//     Standard Inputs/MAIN.R7.T02_STAT/SGs_COM_ERR @bit 1 <-> StandardInputs/Standard Out Var 12
//     Standard Inputs/MAIN.R7.T02_STAT/SGs_COM_ERR <-> StandardInputs/Standard Out Var 9
//     Standard Inputs/MAIN.R7.T02_STAT/SGs_FB_ERR @bit 1 <-> StandardInputs/Standard Out Var 11
//     Standard Inputs/MAIN.R7.T02_STAT/SGs_FB_ERR <-> StandardInputs/Standard Out Var 8
//     Standard Inputs/MAIN.R7.T02_STAT/SGs_OUT_ERR <-> StandardInputs/Standard Out Var 10
//     Standard Inputs/MAIN.R7.T02_STAT/SGs_OUT_ERR @bit 1 <-> StandardInputs/Standard Out Var 13
//     Standard Outputs/MAIN.R7.T02_CMD/FBs_ControlPowerPB <-> StandardOutputs/Standard In Var 7
//     Standard Outputs/MAIN.R7.T02_CMD/SGs_ERRAck <-> StandardOutputs/Standard In Var 4
//     Standard Outputs/MAIN.R7.T02_CMD/SGs_ERRAck <-> StandardOutputs/Standard In Var 6
//     Standard Outputs/MAIN.R7.T02_CMD/SGs_RUNSTOP <-> StandardOutputs/Standard In Var 3
//     Standard Outputs/MAIN.R7.T02_CMD/SGs_RUNSTOP <-> StandardOutputs/Standard In Var 5
//     Standard Outputs/MAIN.Safety_Zone_Test <-> StandardOutputs/Standard In Var 21
//   SODG11_SSCC610_2403701_PLC/SODG11_SSCC610_2403701_PLC Instance <-> EtherCAT Master (EtherCAT)/R7.T01 (EK1100)/R7.T03 (EL1904)
//     Standard Inputs/MAIN.R7.T03/I <-> Module 1 (FSOES)/TxPDO/FSOE/InputChannel1
//     Standard Inputs/MAIN.R7.T03/I @bit 1 <-> Module 1 (FSOES)/TxPDO/FSOE/InputChannel2
//     Standard Inputs/MAIN.R7.T03/I @bit 2 <-> Module 1 (FSOES)/TxPDO/FSOE/InputChannel3
//     Standard Inputs/MAIN.R7.T03/I @bit 3 <-> Module 1 (FSOES)/TxPDO/FSOE/InputChannel4
//     Standard Inputs/MAIN.R7.T03/InfoData/State <-> InfoData/State
//   SODG11_SSCC610_2403701_PLC/SODG11_SSCC610_2403701_PLC Instance <-> EtherCAT Master (EtherCAT)/R7.T01 (EK1100)/R7.T04 (EK1122)
//     Standard Inputs/MAIN.R7.T04/InfoData/State <-> InfoData/State
//   SODG11_SSCC610_2403701_PLC/SODG11_SSCC610_2403701_PLC Instance <-> EtherCAT Master (EtherCAT)/R7.T01 (EK1100)/R7.T04 (EK1122)/R7.Reamer[1].N01 (EP1008-0002)
//     Standard Inputs/MAIN.R7.Reamer[1].N01/I <-> Channel 1/Input
//     Standard Inputs/MAIN.R7.Reamer[1].N01/I @bit 1 <-> Channel 2/Input
//     Standard Inputs/MAIN.R7.Reamer[1].N01/I @bit 2 <-> Channel 3/Input
//     Standard Inputs/MAIN.R7.Reamer[1].N01/I @bit 3 <-> Channel 4/Input
//     Standard Inputs/MAIN.R7.Reamer[1].N01/I @bit 4 <-> Channel 5/Input
//     Standard Inputs/MAIN.R7.Reamer[1].N01/I @bit 5 <-> Channel 6/Input
//     Standard Inputs/MAIN.R7.Reamer[1].N01/I @bit 6 <-> Channel 7/Input
//     Standard Inputs/MAIN.R7.Reamer[1].N01/I @bit 7 <-> Channel 8/Input
//     Standard Inputs/MAIN.R7.Reamer[1].N01/InfoData/State <-> InfoData/State
//     Standard Inputs/MAIN.R7.Reamer[1].N01/Wc_State <-> WcState/WcState
//   SODG11_SSCC610_2403701_PLC/SODG11_SSCC610_2403701_PLC Instance <-> EtherCAT Master (EtherCAT)/R7.T01 (EK1100)/R7.T04 (EK1122)/R7.Reamer[1].N30 (EP2028-0002)
//     Standard Inputs/MAIN.R7.Reamer[1].N30_STAT/InfoData/State <-> InfoData/State
//     Standard Outputs/MAIN.R7.Reamer[1].N30/Q <-> Channel 1/Output
//     Standard Outputs/MAIN.R7.Reamer[1].N30/Q @bit {1..7} <-> Channel {2..8}/Output  (7 links)
//   SODG11_SSCC610_2403701_PLC/SODG11_SSCC610_2403701_PLC Instance <-> EtherCAT Master (EtherCAT)/R8.RT02 (EL6695-1001)
//     Standard Inputs/MAIN.R8.In_From_HW/BYTE_[10] <-> Module 3 (Default IO)/Std. In (64 Bytes)/Input DWORD 2 @bit 8
//     Standard Inputs/MAIN.R8.In_From_HW/BYTE_[11] <-> Module 3 (Default IO)/Std. In (64 Bytes)/Input DWORD 2 @bit 16
//     Standard Inputs/MAIN.R8.In_From_HW/BYTE_[12] <-> Module 3 (Default IO)/Std. In (64 Bytes)/Input DWORD 2 @bit 24
//     Standard Inputs/MAIN.R8.In_From_HW/BYTE_[14] <-> Module 3 (Default IO)/Std. In (64 Bytes)/Input DWORD 3 @bit 8
//     Standard Inputs/MAIN.R8.In_From_HW/BYTE_[15] <-> Module 3 (Default IO)/Std. In (64 Bytes)/Input DWORD 3 @bit 16
//     Standard Inputs/MAIN.R8.In_From_HW/BYTE_[16] <-> Module 3 (Default IO)/Std. In (64 Bytes)/Input DWORD 3 @bit 24
//     Standard Inputs/MAIN.R8.In_From_HW/BYTE_[18] <-> Module 3 (Default IO)/Std. In (64 Bytes)/Input DWORD 4 @bit 8
//     Standard Inputs/MAIN.R8.In_From_HW/BYTE_[19] <-> Module 3 (Default IO)/Std. In (64 Bytes)/Input DWORD 4 @bit 16
//     Standard Inputs/MAIN.R8.In_From_HW/BYTE_[20] <-> Module 3 (Default IO)/Std. In (64 Bytes)/Input DWORD 4 @bit 24
//     Standard Inputs/MAIN.R8.In_From_HW/BYTE_[22] <-> Module 3 (Default IO)/Std. In (64 Bytes)/Input DWORD 5 @bit 8
//     Standard Inputs/MAIN.R8.In_From_HW/BYTE_[23] <-> Module 3 (Default IO)/Std. In (64 Bytes)/Input DWORD 5 @bit 16
//     Standard Inputs/MAIN.R8.In_From_HW/BYTE_[24] <-> Module 3 (Default IO)/Std. In (64 Bytes)/Input DWORD 5 @bit 24
//     Standard Inputs/MAIN.R8.In_From_HW/BYTE_[26] <-> Module 3 (Default IO)/Std. In (64 Bytes)/Input DWORD 6 @bit 8
//     Standard Inputs/MAIN.R8.In_From_HW/BYTE_[27] <-> Module 3 (Default IO)/Std. In (64 Bytes)/Input DWORD 6 @bit 16
//     Standard Inputs/MAIN.R8.In_From_HW/BYTE_[28] <-> Module 3 (Default IO)/Std. In (64 Bytes)/Input DWORD 6 @bit 24
//     Standard Inputs/MAIN.R8.In_From_HW/BYTE_[2] <-> Module 3 (Default IO)/Std. In (64 Bytes)/Input DWORD 0 @bit 8
//     Standard Inputs/MAIN.R8.In_From_HW/BYTE_[30] <-> Module 3 (Default IO)/Std. In (64 Bytes)/Input DWORD 7 @bit 8
//     Standard Inputs/MAIN.R8.In_From_HW/BYTE_[31] <-> Module 3 (Default IO)/Std. In (64 Bytes)/Input DWORD 7 @bit 16
//     Standard Inputs/MAIN.R8.In_From_HW/BYTE_[32] <-> Module 3 (Default IO)/Std. In (64 Bytes)/Input DWORD 7 @bit 24
//     Standard Inputs/MAIN.R8.In_From_HW/BYTE_[34] <-> Module 3 (Default IO)/Std. In (64 Bytes)/Input DWORD 8 @bit 8
//     Standard Inputs/MAIN.R8.In_From_HW/BYTE_[35] <-> Module 3 (Default IO)/Std. In (64 Bytes)/Input DWORD 8 @bit 16
//     Standard Inputs/MAIN.R8.In_From_HW/BYTE_[36] <-> Module 3 (Default IO)/Std. In (64 Bytes)/Input DWORD 8 @bit 24
//     Standard Inputs/MAIN.R8.In_From_HW/BYTE_[38] <-> Module 3 (Default IO)/Std. In (64 Bytes)/Input DWORD 9 @bit 8
//     Standard Inputs/MAIN.R8.In_From_HW/BYTE_[39] <-> Module 3 (Default IO)/Std. In (64 Bytes)/Input DWORD 9 @bit 16
//     Standard Inputs/MAIN.R8.In_From_HW/BYTE_[3] <-> Module 3 (Default IO)/Std. In (64 Bytes)/Input DWORD 0 @bit 16
//     Standard Inputs/MAIN.R8.In_From_HW/BYTE_[40] <-> Module 3 (Default IO)/Std. In (64 Bytes)/Input DWORD 9 @bit 24
//     Standard Inputs/MAIN.R8.In_From_HW/BYTE_[42] <-> Module 3 (Default IO)/Std. In (64 Bytes)/Input DWORD 10 @bit 8
//     Standard Inputs/MAIN.R8.In_From_HW/BYTE_[43] <-> Module 3 (Default IO)/Std. In (64 Bytes)/Input DWORD 10 @bit 16
//     Standard Inputs/MAIN.R8.In_From_HW/BYTE_[44] <-> Module 3 (Default IO)/Std. In (64 Bytes)/Input DWORD 10 @bit 24
//     Standard Inputs/MAIN.R8.In_From_HW/BYTE_[46] <-> Module 3 (Default IO)/Std. In (64 Bytes)/Input DWORD 11 @bit 8
//     Standard Inputs/MAIN.R8.In_From_HW/BYTE_[47] <-> Module 3 (Default IO)/Std. In (64 Bytes)/Input DWORD 11 @bit 16
//     Standard Inputs/MAIN.R8.In_From_HW/BYTE_[48] <-> Module 3 (Default IO)/Std. In (64 Bytes)/Input DWORD 11 @bit 24
//     Standard Inputs/MAIN.R8.In_From_HW/BYTE_[4] <-> Module 3 (Default IO)/Std. In (64 Bytes)/Input DWORD 0 @bit 24
//     Standard Inputs/MAIN.R8.In_From_HW/BYTE_[50] <-> Module 3 (Default IO)/Std. In (64 Bytes)/Input DWORD 12 @bit 8
//     Standard Inputs/MAIN.R8.In_From_HW/BYTE_[51] <-> Module 3 (Default IO)/Std. In (64 Bytes)/Input DWORD 12 @bit 16
//     Standard Inputs/MAIN.R8.In_From_HW/BYTE_[52] <-> Module 3 (Default IO)/Std. In (64 Bytes)/Input DWORD 12 @bit 24
//     Standard Inputs/MAIN.R8.In_From_HW/BYTE_[54] <-> Module 3 (Default IO)/Std. In (64 Bytes)/Input DWORD 13 @bit 8
//     Standard Inputs/MAIN.R8.In_From_HW/BYTE_[55] <-> Module 3 (Default IO)/Std. In (64 Bytes)/Input DWORD 13 @bit 16
//     Standard Inputs/MAIN.R8.In_From_HW/BYTE_[56] <-> Module 3 (Default IO)/Std. In (64 Bytes)/Input DWORD 13 @bit 24
//     Standard Inputs/MAIN.R8.In_From_HW/BYTE_[58] <-> Module 3 (Default IO)/Std. In (64 Bytes)/Input DWORD 14 @bit 8
//     Standard Inputs/MAIN.R8.In_From_HW/BYTE_[59] <-> Module 3 (Default IO)/Std. In (64 Bytes)/Input DWORD 14 @bit 16
//     Standard Inputs/MAIN.R8.In_From_HW/BYTE_[60] <-> Module 3 (Default IO)/Std. In (64 Bytes)/Input DWORD 14 @bit 24
//     Standard Inputs/MAIN.R8.In_From_HW/BYTE_[62] <-> Module 3 (Default IO)/Std. In (64 Bytes)/Input DWORD 15 @bit 8
//     Standard Inputs/MAIN.R8.In_From_HW/BYTE_[63] <-> Module 3 (Default IO)/Std. In (64 Bytes)/Input DWORD 15 @bit 16
//     Standard Inputs/MAIN.R8.In_From_HW/BYTE_[64] <-> Module 3 (Default IO)/Std. In (64 Bytes)/Input DWORD 15 @bit 24
//     Standard Inputs/MAIN.R8.In_From_HW/BYTE_[6] <-> Module 3 (Default IO)/Std. In (64 Bytes)/Input DWORD 1 @bit 8
//     Standard Inputs/MAIN.R8.In_From_HW/BYTE_[7] <-> Module 3 (Default IO)/Std. In (64 Bytes)/Input DWORD 1 @bit 16
//     Standard Inputs/MAIN.R8.In_From_HW/BYTE_[8] <-> Module 3 (Default IO)/Std. In (64 Bytes)/Input DWORD 1 @bit 24
//     Standard Inputs/MAIN.R8.In_From_HW/BYTE_[{1..61 step 4}] <-> Module 3 (Default IO)/Std. In (64 Bytes)/Input DWORD {0..15}  (16 links)
//     Standard Inputs/MAIN.R8.RT02/External_device_not_connected <-> Module 1 (Sync Inputs)/Compact/External device not connected
//     Standard Inputs/MAIN.R8.RT02/FSOE_Inputs_ConnID <-> Module 2 (Safety Data (8 Byte))/Inputs/FSOE/FSOE ConnID
//     Standard Inputs/MAIN.R8.RT02/FSOE_Inputs_Data_0 <-> Module 2 (Safety Data (8 Byte))/Inputs/FSOE/FSOE Data_0
//     Standard Inputs/MAIN.R8.RT02/FSOE_Inputs_Data_1 <-> Module 2 (Safety Data (8 Byte))/Inputs/FSOE/FSOE Data_1
//     Standard Inputs/MAIN.R8.RT02/FSOE_Inputs_Data_2 <-> Module 2 (Safety Data (8 Byte))/Inputs/FSOE/FSOE Data_2
//     Standard Inputs/MAIN.R8.RT02/FSOE_Inputs_Data_3 <-> Module 2 (Safety Data (8 Byte))/Inputs/FSOE/FSOE Data_3
//     Standard Inputs/MAIN.R8.RT02/InfoData/AdsAddr/netId <-> InfoData/AdsAddr/netId
//     Standard Inputs/MAIN.R8.RT02/InfoData/AdsAddr/port <-> InfoData/AdsAddr/port
//     Standard Inputs/MAIN.R8.RT02/InfoData/State <-> InfoData/State
//     Standard Inputs/MAIN.R8.RT02/TxPDO_State <-> Module 1 (Sync Inputs)/Compact/TxPDO state
//     Standard Inputs/MAIN.R8.RT02/TxPDO_Toogle <-> Module 1 (Sync Inputs)/Compact/TxPDO toggle
//     Standard Outputs/MAIN.R8.Out_To_HW/Byte_[10] <-> Module 3 (Default IO)/Std. Out (64 Bytes)/Output DWORD 2 @bit 8
//     Standard Outputs/MAIN.R8.Out_To_HW/Byte_[11] <-> Module 3 (Default IO)/Std. Out (64 Bytes)/Output DWORD 2 @bit 16
//     Standard Outputs/MAIN.R8.Out_To_HW/Byte_[12] <-> Module 3 (Default IO)/Std. Out (64 Bytes)/Output DWORD 2 @bit 24
//     Standard Outputs/MAIN.R8.Out_To_HW/Byte_[14] <-> Module 3 (Default IO)/Std. Out (64 Bytes)/Output DWORD 3 @bit 8
//     Standard Outputs/MAIN.R8.Out_To_HW/Byte_[15] <-> Module 3 (Default IO)/Std. Out (64 Bytes)/Output DWORD 3 @bit 16
//     Standard Outputs/MAIN.R8.Out_To_HW/Byte_[16] <-> Module 3 (Default IO)/Std. Out (64 Bytes)/Output DWORD 3 @bit 24
//     Standard Outputs/MAIN.R8.Out_To_HW/Byte_[18] <-> Module 3 (Default IO)/Std. Out (64 Bytes)/Output DWORD 4 @bit 8
//     Standard Outputs/MAIN.R8.Out_To_HW/Byte_[19] <-> Module 3 (Default IO)/Std. Out (64 Bytes)/Output DWORD 4 @bit 16
//     Standard Outputs/MAIN.R8.Out_To_HW/Byte_[20] <-> Module 3 (Default IO)/Std. Out (64 Bytes)/Output DWORD 4 @bit 24
//     Standard Outputs/MAIN.R8.Out_To_HW/Byte_[22] <-> Module 3 (Default IO)/Std. Out (64 Bytes)/Output DWORD 5 @bit 8
//     Standard Outputs/MAIN.R8.Out_To_HW/Byte_[23] <-> Module 3 (Default IO)/Std. Out (64 Bytes)/Output DWORD 5 @bit 16
//     Standard Outputs/MAIN.R8.Out_To_HW/Byte_[24] <-> Module 3 (Default IO)/Std. Out (64 Bytes)/Output DWORD 5 @bit 24
//     Standard Outputs/MAIN.R8.Out_To_HW/Byte_[26] <-> Module 3 (Default IO)/Std. Out (64 Bytes)/Output DWORD 6 @bit 8
//     Standard Outputs/MAIN.R8.Out_To_HW/Byte_[27] <-> Module 3 (Default IO)/Std. Out (64 Bytes)/Output DWORD 6 @bit 16
//     Standard Outputs/MAIN.R8.Out_To_HW/Byte_[28] <-> Module 3 (Default IO)/Std. Out (64 Bytes)/Output DWORD 6 @bit 24
//     Standard Outputs/MAIN.R8.Out_To_HW/Byte_[2] <-> Module 3 (Default IO)/Std. Out (64 Bytes)/Output DWORD 0 @bit 8
//     Standard Outputs/MAIN.R8.Out_To_HW/Byte_[30] <-> Module 3 (Default IO)/Std. Out (64 Bytes)/Output DWORD 7 @bit 8
//     Standard Outputs/MAIN.R8.Out_To_HW/Byte_[31] <-> Module 3 (Default IO)/Std. Out (64 Bytes)/Output DWORD 7 @bit 16
//     Standard Outputs/MAIN.R8.Out_To_HW/Byte_[32] <-> Module 3 (Default IO)/Std. Out (64 Bytes)/Output DWORD 7 @bit 24
//     Standard Outputs/MAIN.R8.Out_To_HW/Byte_[34] <-> Module 3 (Default IO)/Std. Out (64 Bytes)/Output DWORD 8 @bit 8
//     Standard Outputs/MAIN.R8.Out_To_HW/Byte_[35] <-> Module 3 (Default IO)/Std. Out (64 Bytes)/Output DWORD 8 @bit 16
//     Standard Outputs/MAIN.R8.Out_To_HW/Byte_[36] <-> Module 3 (Default IO)/Std. Out (64 Bytes)/Output DWORD 8 @bit 24
//     Standard Outputs/MAIN.R8.Out_To_HW/Byte_[38] <-> Module 3 (Default IO)/Std. Out (64 Bytes)/Output DWORD 9 @bit 8
//     Standard Outputs/MAIN.R8.Out_To_HW/Byte_[39] <-> Module 3 (Default IO)/Std. Out (64 Bytes)/Output DWORD 9 @bit 16
//     Standard Outputs/MAIN.R8.Out_To_HW/Byte_[3] <-> Module 3 (Default IO)/Std. Out (64 Bytes)/Output DWORD 0 @bit 16
//     Standard Outputs/MAIN.R8.Out_To_HW/Byte_[40] <-> Module 3 (Default IO)/Std. Out (64 Bytes)/Output DWORD 9 @bit 24
//     Standard Outputs/MAIN.R8.Out_To_HW/Byte_[42] <-> Module 3 (Default IO)/Std. Out (64 Bytes)/Output DWORD 10 @bit 8
//     Standard Outputs/MAIN.R8.Out_To_HW/Byte_[43] <-> Module 3 (Default IO)/Std. Out (64 Bytes)/Output DWORD 10 @bit 16
//     Standard Outputs/MAIN.R8.Out_To_HW/Byte_[44] <-> Module 3 (Default IO)/Std. Out (64 Bytes)/Output DWORD 10 @bit 24
//     Standard Outputs/MAIN.R8.Out_To_HW/Byte_[46] <-> Module 3 (Default IO)/Std. Out (64 Bytes)/Output DWORD 11 @bit 8
//     Standard Outputs/MAIN.R8.Out_To_HW/Byte_[47] <-> Module 3 (Default IO)/Std. Out (64 Bytes)/Output DWORD 11 @bit 16
//     Standard Outputs/MAIN.R8.Out_To_HW/Byte_[48] <-> Module 3 (Default IO)/Std. Out (64 Bytes)/Output DWORD 11 @bit 24
//     Standard Outputs/MAIN.R8.Out_To_HW/Byte_[4] <-> Module 3 (Default IO)/Std. Out (64 Bytes)/Output DWORD 0 @bit 24
//     Standard Outputs/MAIN.R8.Out_To_HW/Byte_[50] <-> Module 3 (Default IO)/Std. Out (64 Bytes)/Output DWORD 12 @bit 8
//     Standard Outputs/MAIN.R8.Out_To_HW/Byte_[51] <-> Module 3 (Default IO)/Std. Out (64 Bytes)/Output DWORD 12 @bit 16
//     Standard Outputs/MAIN.R8.Out_To_HW/Byte_[52] <-> Module 3 (Default IO)/Std. Out (64 Bytes)/Output DWORD 12 @bit 24
//     Standard Outputs/MAIN.R8.Out_To_HW/Byte_[54] <-> Module 3 (Default IO)/Std. Out (64 Bytes)/Output DWORD 13 @bit 8
//     Standard Outputs/MAIN.R8.Out_To_HW/Byte_[55] <-> Module 3 (Default IO)/Std. Out (64 Bytes)/Output DWORD 13 @bit 16
//     Standard Outputs/MAIN.R8.Out_To_HW/Byte_[56] <-> Module 3 (Default IO)/Std. Out (64 Bytes)/Output DWORD 13 @bit 24
//     Standard Outputs/MAIN.R8.Out_To_HW/Byte_[58] <-> Module 3 (Default IO)/Std. Out (64 Bytes)/Output DWORD 14 @bit 8
//     Standard Outputs/MAIN.R8.Out_To_HW/Byte_[59] <-> Module 3 (Default IO)/Std. Out (64 Bytes)/Output DWORD 14 @bit 16
//     Standard Outputs/MAIN.R8.Out_To_HW/Byte_[60] <-> Module 3 (Default IO)/Std. Out (64 Bytes)/Output DWORD 14 @bit 24
//     Standard Outputs/MAIN.R8.Out_To_HW/Byte_[62] <-> Module 3 (Default IO)/Std. Out (64 Bytes)/Output DWORD 15 @bit 8
//     Standard Outputs/MAIN.R8.Out_To_HW/Byte_[63] <-> Module 3 (Default IO)/Std. Out (64 Bytes)/Output DWORD 15 @bit 16
//     Standard Outputs/MAIN.R8.Out_To_HW/Byte_[64] <-> Module 3 (Default IO)/Std. Out (64 Bytes)/Output DWORD 15 @bit 24
//     Standard Outputs/MAIN.R8.Out_To_HW/Byte_[6] <-> Module 3 (Default IO)/Std. Out (64 Bytes)/Output DWORD 1 @bit 8
//     Standard Outputs/MAIN.R8.Out_To_HW/Byte_[7] <-> Module 3 (Default IO)/Std. Out (64 Bytes)/Output DWORD 1 @bit 16
//     Standard Outputs/MAIN.R8.Out_To_HW/Byte_[8] <-> Module 3 (Default IO)/Std. Out (64 Bytes)/Output DWORD 1 @bit 24
//     Standard Outputs/MAIN.R8.Out_To_HW/Byte_[{1..61 step 4}] <-> Module 3 (Default IO)/Std. Out (64 Bytes)/Output DWORD {0..15}  (16 links)
//   SODG11_SSCC610_2403701_PLC/SODG11_SSCC610_2403701_PLC Instance <-> EtherCAT Master (EtherCAT)/R8.T01 (EK1100)
//     Standard Inputs/MAIN.R8.T01/InfoData/State <-> InfoData/State
//   SODG11_SSCC610_2403701_PLC/SODG11_SSCC610_2403701_PLC Instance <-> EtherCAT Master (EtherCAT)/R8.T01 (EK1100)/R8.T02 (EL6900)
//     Standard Inputs/MAIN.R8.RT02/FSOE_Outputs_Data_0 @bit 1 <-> StandardInputs/Standard Out Var 14
//     Standard Inputs/MAIN.R8.RT02/FSOE_Outputs_Data_0 @bit 2 <-> StandardInputs/Standard Out Var 15
//     Standard Inputs/MAIN.R8.RT02/FSOE_Outputs_Data_2 @bit 1 <-> StandardInputs/Standard Out Var 18
//     Standard Inputs/MAIN.R8.RT02/FSOE_Outputs_Data_2 <-> StandardInputs/Standard Out Var 17
//     Standard Inputs/MAIN.R8.T02_STAT/Device_Info_Data/Project_CRC <-> Device Info Data/Project CRC
//     Standard Inputs/MAIN.R8.T02_STAT/FBs_FB_ERR <-> StandardInputs/Standard Out Var 16
//     Standard Inputs/MAIN.R8.T02_STAT/FBs_FB_ERR @bit 16 <-> StandardInputs/Standard Out Var 19
//     Standard Inputs/MAIN.R8.T02_STAT/FBs_FB_ERR @bit 29 <-> StandardInputs/Standard Out Var 20
//     Standard Inputs/MAIN.R8.T02_STAT/InfoData/AdsAddr/netId <-> InfoData/AdsAddr/netId
//     Standard Inputs/MAIN.R8.T02_STAT/InfoData/AdsAddr/port <-> InfoData/AdsAddr/port
//     Standard Inputs/MAIN.R8.T02_STAT/InfoData/State <-> InfoData/State
//     Standard Inputs/MAIN.R8.T02_STAT/SGs_COM_ERR @bit 1 <-> StandardInputs/Standard Out Var 12
//     Standard Inputs/MAIN.R8.T02_STAT/SGs_COM_ERR <-> StandardInputs/Standard Out Var 9
//     Standard Inputs/MAIN.R8.T02_STAT/SGs_FB_ERR @bit 1 <-> StandardInputs/Standard Out Var 11
//     Standard Inputs/MAIN.R8.T02_STAT/SGs_FB_ERR <-> StandardInputs/Standard Out Var 8
//     Standard Inputs/MAIN.R8.T02_STAT/SGs_OUT_ERR <-> StandardInputs/Standard Out Var 10
//     Standard Inputs/MAIN.R8.T02_STAT/SGs_OUT_ERR @bit 1 <-> StandardInputs/Standard Out Var 13
//     Standard Outputs/MAIN.R8.T02_CMD/FBs_ControlPowerPB <-> StandardOutputs/Standard In Var 7
//     Standard Outputs/MAIN.R8.T02_CMD/SGs_ERRAck <-> StandardOutputs/Standard In Var 4
//     Standard Outputs/MAIN.R8.T02_CMD/SGs_ERRAck <-> StandardOutputs/Standard In Var 6
//     Standard Outputs/MAIN.R8.T02_CMD/SGs_RUNSTOP <-> StandardOutputs/Standard In Var 3
//     Standard Outputs/MAIN.R8.T02_CMD/SGs_RUNSTOP <-> StandardOutputs/Standard In Var 5
//     Standard Outputs/MAIN.Safety_Zone_Test <-> StandardOutputs/Standard In Var 21
//   SODG11_SSCC610_2403701_PLC/SODG11_SSCC610_2403701_PLC Instance <-> EtherCAT Master (EtherCAT)/R8.T01 (EK1100)/R8.T03 (EL1904)
//     Standard Inputs/MAIN.R8.T03/I <-> Module 1 (FSOES)/TxPDO/FSOE/InputChannel1
//     Standard Inputs/MAIN.R8.T03/I @bit 1 <-> Module 1 (FSOES)/TxPDO/FSOE/InputChannel2
//     Standard Inputs/MAIN.R8.T03/I @bit 2 <-> Module 1 (FSOES)/TxPDO/FSOE/InputChannel3
//     Standard Inputs/MAIN.R8.T03/I @bit 3 <-> Module 1 (FSOES)/TxPDO/FSOE/InputChannel4
//     Standard Inputs/MAIN.R8.T03/InfoData/State <-> InfoData/State
//   SODG11_SSCC610_2403701_PLC/SODG11_SSCC610_2403701_PLC Instance <-> EtherCAT Master (EtherCAT)/R8.T01 (EK1100)/R8.T04 (EK1122)
//     Standard Inputs/MAIN.R8.T04/InfoData/State <-> InfoData/State
//   SODG11_SSCC610_2403701_PLC/SODG11_SSCC610_2403701_PLC Instance <-> EtherCAT Master (EtherCAT)/R8.T01 (EK1100)/R8.T04 (EK1122)/R8.Reamer[1].N01 (EP1008-0002)
//     Standard Inputs/MAIN.R8.Reamer[1].N01/I <-> Channel 1/Input
//     Standard Inputs/MAIN.R8.Reamer[1].N01/I @bit 1 <-> Channel 2/Input
//     Standard Inputs/MAIN.R8.Reamer[1].N01/I @bit 2 <-> Channel 3/Input
//     Standard Inputs/MAIN.R8.Reamer[1].N01/I @bit 3 <-> Channel 4/Input
//     Standard Inputs/MAIN.R8.Reamer[1].N01/I @bit 4 <-> Channel 5/Input
//     Standard Inputs/MAIN.R8.Reamer[1].N01/I @bit 5 <-> Channel 6/Input
//     Standard Inputs/MAIN.R8.Reamer[1].N01/I @bit 6 <-> Channel 7/Input
//     Standard Inputs/MAIN.R8.Reamer[1].N01/I @bit 7 <-> Channel 8/Input
//     Standard Inputs/MAIN.R8.Reamer[1].N01/InfoData/State <-> InfoData/State
//     Standard Inputs/MAIN.R8.Reamer[1].N01/Wc_State <-> WcState/WcState
//   SODG11_SSCC610_2403701_PLC/SODG11_SSCC610_2403701_PLC Instance <-> EtherCAT Master (EtherCAT)/R8.T01 (EK1100)/R8.T04 (EK1122)/R8.Reamer[1].N30 (EP2028-0002)
//     Standard Inputs/MAIN.R8.Reamer[1].N30_STAT/InfoData/State <-> InfoData/State
//     Standard Outputs/MAIN.R8.Reamer[1].N30/Q <-> Channel 1/Output
//     Standard Outputs/MAIN.R8.Reamer[1].N30/Q @bit {1..7} <-> Channel {2..8}/Output  (7 links)
//   SODG11_SSCC610_2403701_PLC/SODG11_SSCC610_2403701_PLC Instance <-> EtherCAT Master (EtherCAT)/R9.RT02 (EL6695-1001)
//     Standard Inputs/MAIN.R9.In_From_HW/BYTE_[10] <-> Module 3 (Default IO)/Std. In (64 Bytes)/Input DWORD 2 @bit 8
//     Standard Inputs/MAIN.R9.In_From_HW/BYTE_[11] <-> Module 3 (Default IO)/Std. In (64 Bytes)/Input DWORD 2 @bit 16
//     Standard Inputs/MAIN.R9.In_From_HW/BYTE_[12] <-> Module 3 (Default IO)/Std. In (64 Bytes)/Input DWORD 2 @bit 24
//     Standard Inputs/MAIN.R9.In_From_HW/BYTE_[14] <-> Module 3 (Default IO)/Std. In (64 Bytes)/Input DWORD 3 @bit 8
//     Standard Inputs/MAIN.R9.In_From_HW/BYTE_[15] <-> Module 3 (Default IO)/Std. In (64 Bytes)/Input DWORD 3 @bit 16
//     Standard Inputs/MAIN.R9.In_From_HW/BYTE_[16] <-> Module 3 (Default IO)/Std. In (64 Bytes)/Input DWORD 3 @bit 24
//     Standard Inputs/MAIN.R9.In_From_HW/BYTE_[18] <-> Module 3 (Default IO)/Std. In (64 Bytes)/Input DWORD 4 @bit 8
//     Standard Inputs/MAIN.R9.In_From_HW/BYTE_[19] <-> Module 3 (Default IO)/Std. In (64 Bytes)/Input DWORD 4 @bit 16
//     Standard Inputs/MAIN.R9.In_From_HW/BYTE_[20] <-> Module 3 (Default IO)/Std. In (64 Bytes)/Input DWORD 4 @bit 24
//     Standard Inputs/MAIN.R9.In_From_HW/BYTE_[22] <-> Module 3 (Default IO)/Std. In (64 Bytes)/Input DWORD 5 @bit 8
//     Standard Inputs/MAIN.R9.In_From_HW/BYTE_[23] <-> Module 3 (Default IO)/Std. In (64 Bytes)/Input DWORD 5 @bit 16
//     Standard Inputs/MAIN.R9.In_From_HW/BYTE_[24] <-> Module 3 (Default IO)/Std. In (64 Bytes)/Input DWORD 5 @bit 24
//     Standard Inputs/MAIN.R9.In_From_HW/BYTE_[26] <-> Module 3 (Default IO)/Std. In (64 Bytes)/Input DWORD 6 @bit 8
//     Standard Inputs/MAIN.R9.In_From_HW/BYTE_[27] <-> Module 3 (Default IO)/Std. In (64 Bytes)/Input DWORD 6 @bit 16
//     Standard Inputs/MAIN.R9.In_From_HW/BYTE_[28] <-> Module 3 (Default IO)/Std. In (64 Bytes)/Input DWORD 6 @bit 24
//     Standard Inputs/MAIN.R9.In_From_HW/BYTE_[2] <-> Module 3 (Default IO)/Std. In (64 Bytes)/Input DWORD 0 @bit 8
//     Standard Inputs/MAIN.R9.In_From_HW/BYTE_[30] <-> Module 3 (Default IO)/Std. In (64 Bytes)/Input DWORD 7 @bit 8
//     Standard Inputs/MAIN.R9.In_From_HW/BYTE_[31] <-> Module 3 (Default IO)/Std. In (64 Bytes)/Input DWORD 7 @bit 16
//     Standard Inputs/MAIN.R9.In_From_HW/BYTE_[32] <-> Module 3 (Default IO)/Std. In (64 Bytes)/Input DWORD 7 @bit 24
//     Standard Inputs/MAIN.R9.In_From_HW/BYTE_[34] <-> Module 3 (Default IO)/Std. In (64 Bytes)/Input DWORD 8 @bit 8
//     Standard Inputs/MAIN.R9.In_From_HW/BYTE_[35] <-> Module 3 (Default IO)/Std. In (64 Bytes)/Input DWORD 8 @bit 16
//     Standard Inputs/MAIN.R9.In_From_HW/BYTE_[36] <-> Module 3 (Default IO)/Std. In (64 Bytes)/Input DWORD 8 @bit 24
//     Standard Inputs/MAIN.R9.In_From_HW/BYTE_[38] <-> Module 3 (Default IO)/Std. In (64 Bytes)/Input DWORD 9 @bit 8
//     Standard Inputs/MAIN.R9.In_From_HW/BYTE_[39] <-> Module 3 (Default IO)/Std. In (64 Bytes)/Input DWORD 9 @bit 16
//     Standard Inputs/MAIN.R9.In_From_HW/BYTE_[3] <-> Module 3 (Default IO)/Std. In (64 Bytes)/Input DWORD 0 @bit 16
//     Standard Inputs/MAIN.R9.In_From_HW/BYTE_[40] <-> Module 3 (Default IO)/Std. In (64 Bytes)/Input DWORD 9 @bit 24
//     Standard Inputs/MAIN.R9.In_From_HW/BYTE_[42] <-> Module 3 (Default IO)/Std. In (64 Bytes)/Input DWORD 10 @bit 8
//     Standard Inputs/MAIN.R9.In_From_HW/BYTE_[43] <-> Module 3 (Default IO)/Std. In (64 Bytes)/Input DWORD 10 @bit 16
//     Standard Inputs/MAIN.R9.In_From_HW/BYTE_[44] <-> Module 3 (Default IO)/Std. In (64 Bytes)/Input DWORD 10 @bit 24
//     Standard Inputs/MAIN.R9.In_From_HW/BYTE_[46] <-> Module 3 (Default IO)/Std. In (64 Bytes)/Input DWORD 11 @bit 8
//     Standard Inputs/MAIN.R9.In_From_HW/BYTE_[47] <-> Module 3 (Default IO)/Std. In (64 Bytes)/Input DWORD 11 @bit 16
//     Standard Inputs/MAIN.R9.In_From_HW/BYTE_[48] <-> Module 3 (Default IO)/Std. In (64 Bytes)/Input DWORD 11 @bit 24
//     Standard Inputs/MAIN.R9.In_From_HW/BYTE_[4] <-> Module 3 (Default IO)/Std. In (64 Bytes)/Input DWORD 0 @bit 24
//     Standard Inputs/MAIN.R9.In_From_HW/BYTE_[50] <-> Module 3 (Default IO)/Std. In (64 Bytes)/Input DWORD 12 @bit 8
//     Standard Inputs/MAIN.R9.In_From_HW/BYTE_[51] <-> Module 3 (Default IO)/Std. In (64 Bytes)/Input DWORD 12 @bit 16
//     Standard Inputs/MAIN.R9.In_From_HW/BYTE_[52] <-> Module 3 (Default IO)/Std. In (64 Bytes)/Input DWORD 12 @bit 24
//     Standard Inputs/MAIN.R9.In_From_HW/BYTE_[54] <-> Module 3 (Default IO)/Std. In (64 Bytes)/Input DWORD 13 @bit 8
//     Standard Inputs/MAIN.R9.In_From_HW/BYTE_[55] <-> Module 3 (Default IO)/Std. In (64 Bytes)/Input DWORD 13 @bit 16
//     Standard Inputs/MAIN.R9.In_From_HW/BYTE_[56] <-> Module 3 (Default IO)/Std. In (64 Bytes)/Input DWORD 13 @bit 24
//     Standard Inputs/MAIN.R9.In_From_HW/BYTE_[58] <-> Module 3 (Default IO)/Std. In (64 Bytes)/Input DWORD 14 @bit 8
//     Standard Inputs/MAIN.R9.In_From_HW/BYTE_[59] <-> Module 3 (Default IO)/Std. In (64 Bytes)/Input DWORD 14 @bit 16
//     Standard Inputs/MAIN.R9.In_From_HW/BYTE_[60] <-> Module 3 (Default IO)/Std. In (64 Bytes)/Input DWORD 14 @bit 24
//     Standard Inputs/MAIN.R9.In_From_HW/BYTE_[62] <-> Module 3 (Default IO)/Std. In (64 Bytes)/Input DWORD 15 @bit 8
//     Standard Inputs/MAIN.R9.In_From_HW/BYTE_[63] <-> Module 3 (Default IO)/Std. In (64 Bytes)/Input DWORD 15 @bit 16
//     Standard Inputs/MAIN.R9.In_From_HW/BYTE_[64] <-> Module 3 (Default IO)/Std. In (64 Bytes)/Input DWORD 15 @bit 24
//     Standard Inputs/MAIN.R9.In_From_HW/BYTE_[6] <-> Module 3 (Default IO)/Std. In (64 Bytes)/Input DWORD 1 @bit 8
//     Standard Inputs/MAIN.R9.In_From_HW/BYTE_[7] <-> Module 3 (Default IO)/Std. In (64 Bytes)/Input DWORD 1 @bit 16
//     Standard Inputs/MAIN.R9.In_From_HW/BYTE_[8] <-> Module 3 (Default IO)/Std. In (64 Bytes)/Input DWORD 1 @bit 24
//     Standard Inputs/MAIN.R9.In_From_HW/BYTE_[{1..61 step 4}] <-> Module 3 (Default IO)/Std. In (64 Bytes)/Input DWORD {0..15}  (16 links)
//     Standard Inputs/MAIN.R9.RT02/External_device_not_connected <-> Module 1 (Sync Inputs)/Compact/External device not connected
//     Standard Inputs/MAIN.R9.RT02/FSOE_Inputs_ConnID <-> Module 2 (Safety Data (8 Byte))/Inputs/FSOE/FSOE ConnID
//     Standard Inputs/MAIN.R9.RT02/FSOE_Inputs_Data_0 <-> Module 2 (Safety Data (8 Byte))/Inputs/FSOE/FSOE Data_0
//     Standard Inputs/MAIN.R9.RT02/FSOE_Inputs_Data_1 <-> Module 2 (Safety Data (8 Byte))/Inputs/FSOE/FSOE Data_1
//     Standard Inputs/MAIN.R9.RT02/FSOE_Inputs_Data_2 <-> Module 2 (Safety Data (8 Byte))/Inputs/FSOE/FSOE Data_2
//     Standard Inputs/MAIN.R9.RT02/FSOE_Inputs_Data_3 <-> Module 2 (Safety Data (8 Byte))/Inputs/FSOE/FSOE Data_3
//     Standard Inputs/MAIN.R9.RT02/InfoData/AdsAddr/netId <-> InfoData/AdsAddr/netId
//     Standard Inputs/MAIN.R9.RT02/InfoData/AdsAddr/port <-> InfoData/AdsAddr/port
//     Standard Inputs/MAIN.R9.RT02/InfoData/State <-> InfoData/State
//     Standard Inputs/MAIN.R9.RT02/TxPDO_State <-> Module 1 (Sync Inputs)/Compact/TxPDO state
//     Standard Inputs/MAIN.R9.RT02/TxPDO_Toogle <-> Module 1 (Sync Inputs)/Compact/TxPDO toggle
//     Standard Outputs/MAIN.R9.Out_To_HW/Byte_[10] <-> Module 3 (Default IO)/Std. Out (64 Bytes)/Output DWORD 2 @bit 8
//     Standard Outputs/MAIN.R9.Out_To_HW/Byte_[11] <-> Module 3 (Default IO)/Std. Out (64 Bytes)/Output DWORD 2 @bit 16
//     Standard Outputs/MAIN.R9.Out_To_HW/Byte_[12] <-> Module 3 (Default IO)/Std. Out (64 Bytes)/Output DWORD 2 @bit 24
//     Standard Outputs/MAIN.R9.Out_To_HW/Byte_[14] <-> Module 3 (Default IO)/Std. Out (64 Bytes)/Output DWORD 3 @bit 8
//     Standard Outputs/MAIN.R9.Out_To_HW/Byte_[15] <-> Module 3 (Default IO)/Std. Out (64 Bytes)/Output DWORD 3 @bit 16
//     Standard Outputs/MAIN.R9.Out_To_HW/Byte_[16] <-> Module 3 (Default IO)/Std. Out (64 Bytes)/Output DWORD 3 @bit 24
//     Standard Outputs/MAIN.R9.Out_To_HW/Byte_[18] <-> Module 3 (Default IO)/Std. Out (64 Bytes)/Output DWORD 4 @bit 8
//     Standard Outputs/MAIN.R9.Out_To_HW/Byte_[19] <-> Module 3 (Default IO)/Std. Out (64 Bytes)/Output DWORD 4 @bit 16
//     Standard Outputs/MAIN.R9.Out_To_HW/Byte_[20] <-> Module 3 (Default IO)/Std. Out (64 Bytes)/Output DWORD 4 @bit 24
//     Standard Outputs/MAIN.R9.Out_To_HW/Byte_[22] <-> Module 3 (Default IO)/Std. Out (64 Bytes)/Output DWORD 5 @bit 8
//     Standard Outputs/MAIN.R9.Out_To_HW/Byte_[23] <-> Module 3 (Default IO)/Std. Out (64 Bytes)/Output DWORD 5 @bit 16
//     Standard Outputs/MAIN.R9.Out_To_HW/Byte_[24] <-> Module 3 (Default IO)/Std. Out (64 Bytes)/Output DWORD 5 @bit 24
//     Standard Outputs/MAIN.R9.Out_To_HW/Byte_[26] <-> Module 3 (Default IO)/Std. Out (64 Bytes)/Output DWORD 6 @bit 8
//     Standard Outputs/MAIN.R9.Out_To_HW/Byte_[27] <-> Module 3 (Default IO)/Std. Out (64 Bytes)/Output DWORD 6 @bit 16
//     Standard Outputs/MAIN.R9.Out_To_HW/Byte_[28] <-> Module 3 (Default IO)/Std. Out (64 Bytes)/Output DWORD 6 @bit 24
//     Standard Outputs/MAIN.R9.Out_To_HW/Byte_[2] <-> Module 3 (Default IO)/Std. Out (64 Bytes)/Output DWORD 0 @bit 8
//     Standard Outputs/MAIN.R9.Out_To_HW/Byte_[30] <-> Module 3 (Default IO)/Std. Out (64 Bytes)/Output DWORD 7 @bit 8
//     Standard Outputs/MAIN.R9.Out_To_HW/Byte_[31] <-> Module 3 (Default IO)/Std. Out (64 Bytes)/Output DWORD 7 @bit 16
//     Standard Outputs/MAIN.R9.Out_To_HW/Byte_[32] <-> Module 3 (Default IO)/Std. Out (64 Bytes)/Output DWORD 7 @bit 24
//     Standard Outputs/MAIN.R9.Out_To_HW/Byte_[34] <-> Module 3 (Default IO)/Std. Out (64 Bytes)/Output DWORD 8 @bit 8
//     Standard Outputs/MAIN.R9.Out_To_HW/Byte_[35] <-> Module 3 (Default IO)/Std. Out (64 Bytes)/Output DWORD 8 @bit 16
//     Standard Outputs/MAIN.R9.Out_To_HW/Byte_[36] <-> Module 3 (Default IO)/Std. Out (64 Bytes)/Output DWORD 8 @bit 24
//     Standard Outputs/MAIN.R9.Out_To_HW/Byte_[38] <-> Module 3 (Default IO)/Std. Out (64 Bytes)/Output DWORD 9 @bit 8
//     Standard Outputs/MAIN.R9.Out_To_HW/Byte_[39] <-> Module 3 (Default IO)/Std. Out (64 Bytes)/Output DWORD 9 @bit 16
//     Standard Outputs/MAIN.R9.Out_To_HW/Byte_[3] <-> Module 3 (Default IO)/Std. Out (64 Bytes)/Output DWORD 0 @bit 16
//     Standard Outputs/MAIN.R9.Out_To_HW/Byte_[40] <-> Module 3 (Default IO)/Std. Out (64 Bytes)/Output DWORD 9 @bit 24
//     Standard Outputs/MAIN.R9.Out_To_HW/Byte_[42] <-> Module 3 (Default IO)/Std. Out (64 Bytes)/Output DWORD 10 @bit 8
//     Standard Outputs/MAIN.R9.Out_To_HW/Byte_[43] <-> Module 3 (Default IO)/Std. Out (64 Bytes)/Output DWORD 10 @bit 16
//     Standard Outputs/MAIN.R9.Out_To_HW/Byte_[44] <-> Module 3 (Default IO)/Std. Out (64 Bytes)/Output DWORD 10 @bit 24
//     Standard Outputs/MAIN.R9.Out_To_HW/Byte_[46] <-> Module 3 (Default IO)/Std. Out (64 Bytes)/Output DWORD 11 @bit 8
//     Standard Outputs/MAIN.R9.Out_To_HW/Byte_[47] <-> Module 3 (Default IO)/Std. Out (64 Bytes)/Output DWORD 11 @bit 16
//     Standard Outputs/MAIN.R9.Out_To_HW/Byte_[48] <-> Module 3 (Default IO)/Std. Out (64 Bytes)/Output DWORD 11 @bit 24
//     Standard Outputs/MAIN.R9.Out_To_HW/Byte_[4] <-> Module 3 (Default IO)/Std. Out (64 Bytes)/Output DWORD 0 @bit 24
//     Standard Outputs/MAIN.R9.Out_To_HW/Byte_[50] <-> Module 3 (Default IO)/Std. Out (64 Bytes)/Output DWORD 12 @bit 8
//     Standard Outputs/MAIN.R9.Out_To_HW/Byte_[51] <-> Module 3 (Default IO)/Std. Out (64 Bytes)/Output DWORD 12 @bit 16
//     Standard Outputs/MAIN.R9.Out_To_HW/Byte_[52] <-> Module 3 (Default IO)/Std. Out (64 Bytes)/Output DWORD 12 @bit 24
//     Standard Outputs/MAIN.R9.Out_To_HW/Byte_[54] <-> Module 3 (Default IO)/Std. Out (64 Bytes)/Output DWORD 13 @bit 8
//     Standard Outputs/MAIN.R9.Out_To_HW/Byte_[55] <-> Module 3 (Default IO)/Std. Out (64 Bytes)/Output DWORD 13 @bit 16
//     Standard Outputs/MAIN.R9.Out_To_HW/Byte_[56] <-> Module 3 (Default IO)/Std. Out (64 Bytes)/Output DWORD 13 @bit 24
//     Standard Outputs/MAIN.R9.Out_To_HW/Byte_[58] <-> Module 3 (Default IO)/Std. Out (64 Bytes)/Output DWORD 14 @bit 8
//     Standard Outputs/MAIN.R9.Out_To_HW/Byte_[59] <-> Module 3 (Default IO)/Std. Out (64 Bytes)/Output DWORD 14 @bit 16
//     Standard Outputs/MAIN.R9.Out_To_HW/Byte_[60] <-> Module 3 (Default IO)/Std. Out (64 Bytes)/Output DWORD 14 @bit 24
//     Standard Outputs/MAIN.R9.Out_To_HW/Byte_[62] <-> Module 3 (Default IO)/Std. Out (64 Bytes)/Output DWORD 15 @bit 8
//     Standard Outputs/MAIN.R9.Out_To_HW/Byte_[63] <-> Module 3 (Default IO)/Std. Out (64 Bytes)/Output DWORD 15 @bit 16
//     Standard Outputs/MAIN.R9.Out_To_HW/Byte_[64] <-> Module 3 (Default IO)/Std. Out (64 Bytes)/Output DWORD 15 @bit 24
//     Standard Outputs/MAIN.R9.Out_To_HW/Byte_[6] <-> Module 3 (Default IO)/Std. Out (64 Bytes)/Output DWORD 1 @bit 8
//     Standard Outputs/MAIN.R9.Out_To_HW/Byte_[7] <-> Module 3 (Default IO)/Std. Out (64 Bytes)/Output DWORD 1 @bit 16
//     Standard Outputs/MAIN.R9.Out_To_HW/Byte_[8] <-> Module 3 (Default IO)/Std. Out (64 Bytes)/Output DWORD 1 @bit 24
//     Standard Outputs/MAIN.R9.Out_To_HW/Byte_[{1..61 step 4}] <-> Module 3 (Default IO)/Std. Out (64 Bytes)/Output DWORD {0..15}  (16 links)
//   SODG11_SSCC610_2403701_PLC/SODG11_SSCC610_2403701_PLC Instance <-> EtherCAT Master (EtherCAT)/R9.T01 (EK1100)
//     Standard Inputs/MAIN.R9.T01/InfoData/State <-> InfoData/State
//   SODG11_SSCC610_2403701_PLC/SODG11_SSCC610_2403701_PLC Instance <-> EtherCAT Master (EtherCAT)/R9.T01 (EK1100)/R9.T02 (EL6900)
//     Standard Inputs/MAIN.R9.RT02/FSOE_Outputs_Data_0 @bit 1 <-> StandardInputs/Standard Out Var 14
//     Standard Inputs/MAIN.R9.RT02/FSOE_Outputs_Data_0 @bit 2 <-> StandardInputs/Standard Out Var 15
//     Standard Inputs/MAIN.R9.RT02/FSOE_Outputs_Data_2 @bit 1 <-> StandardInputs/Standard Out Var 18
//     Standard Inputs/MAIN.R9.RT02/FSOE_Outputs_Data_2 <-> StandardInputs/Standard Out Var 17
//     Standard Inputs/MAIN.R9.T02_STAT/Device_Info_Data/Project_CRC <-> Device Info Data/Project CRC
//     Standard Inputs/MAIN.R9.T02_STAT/FBs_FB_ERR <-> StandardInputs/Standard Out Var 16
//     Standard Inputs/MAIN.R9.T02_STAT/FBs_FB_ERR @bit 16 <-> StandardInputs/Standard Out Var 19
//     Standard Inputs/MAIN.R9.T02_STAT/FBs_FB_ERR @bit 29 <-> StandardInputs/Standard Out Var 20
//     Standard Inputs/MAIN.R9.T02_STAT/InfoData/AdsAddr/netId <-> InfoData/AdsAddr/netId
//     Standard Inputs/MAIN.R9.T02_STAT/InfoData/AdsAddr/port <-> InfoData/AdsAddr/port
//     Standard Inputs/MAIN.R9.T02_STAT/InfoData/State <-> InfoData/State
//     Standard Inputs/MAIN.R9.T02_STAT/SGs_COM_ERR @bit 1 <-> StandardInputs/Standard Out Var 12
//     Standard Inputs/MAIN.R9.T02_STAT/SGs_COM_ERR <-> StandardInputs/Standard Out Var 9
//     Standard Inputs/MAIN.R9.T02_STAT/SGs_FB_ERR @bit 1 <-> StandardInputs/Standard Out Var 11
//     Standard Inputs/MAIN.R9.T02_STAT/SGs_FB_ERR <-> StandardInputs/Standard Out Var 8
//     Standard Inputs/MAIN.R9.T02_STAT/SGs_OUT_ERR <-> StandardInputs/Standard Out Var 10
//     Standard Inputs/MAIN.R9.T02_STAT/SGs_OUT_ERR @bit 1 <-> StandardInputs/Standard Out Var 13
//     Standard Outputs/MAIN.R9.T02_CMD/FBs_ControlPowerPB <-> StandardOutputs/Standard In Var 7
//     Standard Outputs/MAIN.R9.T02_CMD/SGs_ERRAck <-> StandardOutputs/Standard In Var 4
//     Standard Outputs/MAIN.R9.T02_CMD/SGs_ERRAck <-> StandardOutputs/Standard In Var 6
//     Standard Outputs/MAIN.R9.T02_CMD/SGs_RUNSTOP <-> StandardOutputs/Standard In Var 3
//     Standard Outputs/MAIN.R9.T02_CMD/SGs_RUNSTOP <-> StandardOutputs/Standard In Var 5
//     Standard Outputs/MAIN.Safety_Zone_Test <-> StandardOutputs/Standard In Var 21
//   SODG11_SSCC610_2403701_PLC/SODG11_SSCC610_2403701_PLC Instance <-> EtherCAT Master (EtherCAT)/R9.T01 (EK1100)/R9.T03 (EL1904)
//     Standard Inputs/MAIN.R9.T03/I <-> Module 1 (FSOES)/TxPDO/FSOE/InputChannel1
//     Standard Inputs/MAIN.R9.T03/I @bit 1 <-> Module 1 (FSOES)/TxPDO/FSOE/InputChannel2
//     Standard Inputs/MAIN.R9.T03/I @bit 2 <-> Module 1 (FSOES)/TxPDO/FSOE/InputChannel3
//     Standard Inputs/MAIN.R9.T03/I @bit 3 <-> Module 1 (FSOES)/TxPDO/FSOE/InputChannel4
//     Standard Inputs/MAIN.R9.T03/InfoData/State <-> InfoData/State
//   SODG11_SSCC610_2403701_PLC/SODG11_SSCC610_2403701_PLC Instance <-> EtherCAT Master (EtherCAT)/R9.T01 (EK1100)/R9.T04 (EK1122)
//     Standard Inputs/MAIN.R9.T04/InfoData/State <-> InfoData/State
//   SODG11_SSCC610_2403701_PLC/SODG11_SSCC610_2403701_PLC Instance <-> EtherCAT Master (EtherCAT)/R9.T01 (EK1100)/R9.T04 (EK1122)/R9.Reamer[1].N01 (EP1008-0002)
//     Standard Inputs/MAIN.R9.Reamer[1].N01/I <-> Channel 1/Input
//     Standard Inputs/MAIN.R9.Reamer[1].N01/I @bit 1 <-> Channel 2/Input
//     Standard Inputs/MAIN.R9.Reamer[1].N01/I @bit 2 <-> Channel 3/Input
//     Standard Inputs/MAIN.R9.Reamer[1].N01/I @bit 3 <-> Channel 4/Input
//     Standard Inputs/MAIN.R9.Reamer[1].N01/I @bit 4 <-> Channel 5/Input
//     Standard Inputs/MAIN.R9.Reamer[1].N01/I @bit 5 <-> Channel 6/Input
//     Standard Inputs/MAIN.R9.Reamer[1].N01/I @bit 6 <-> Channel 7/Input
//     Standard Inputs/MAIN.R9.Reamer[1].N01/I @bit 7 <-> Channel 8/Input
//     Standard Inputs/MAIN.R9.Reamer[1].N01/InfoData/State <-> InfoData/State
//     Standard Inputs/MAIN.R9.Reamer[1].N01/Wc_State <-> WcState/WcState
//   SODG11_SSCC610_2403701_PLC/SODG11_SSCC610_2403701_PLC Instance <-> EtherCAT Master (EtherCAT)/R9.T01 (EK1100)/R9.T04 (EK1122)/R9.Reamer[1].N30 (EP2028-0002)
//     Standard Inputs/MAIN.R9.Reamer[1].N30_STAT/InfoData/State <-> InfoData/State
//     Standard Outputs/MAIN.R9.Reamer[1].N30/Q <-> Channel 1/Output
//     Standard Outputs/MAIN.R9.Reamer[1].N30/Q @bit {1..7} <-> Channel {2..8}/Output  (7 links)
//   SODG11_SSCC610_2403701_PLC/SODG11_SSCC610_2403701_PLC Instance <-> EtherCAT Master (EtherCAT)/SS01.N01 (EP9128-0021)
//     Standard Inputs/MAIN.IS01.N01/InfoData/State <-> InfoData/State
//     Standard Inputs/MAIN.SS01.N01/InfoData/State <-> InfoData/State
//   SODG11_SSCC610_2403701_PLC/SODG11_SSCC610_2403701_PLC Instance <-> EtherCAT Master (EtherCAT)/SS01.N01 (EP9128-0021)/Fix101.N01 (EP1008-0002)
//     Standard Inputs/Fix101.N01/I <-> Channel 1/Input
//     Standard Inputs/Fix101.N01/I @bit 1 <-> Channel 2/Input
//     Standard Inputs/Fix101.N01/I @bit 2 <-> Channel 3/Input
//     Standard Inputs/Fix101.N01/I @bit 3 <-> Channel 4/Input
//     Standard Inputs/Fix101.N01/I @bit 4 <-> Channel 5/Input
//     Standard Inputs/Fix101.N01/I @bit 5 <-> Channel 6/Input
//     Standard Inputs/Fix101.N01/I @bit 6 <-> Channel 7/Input
//     Standard Inputs/Fix101.N01/I @bit 7 <-> Channel 8/Input
//     Standard Inputs/Fix101.N01/InfoData/State <-> InfoData/State
//     Standard Inputs/Fix101.N01/Wc_State <-> WcState/WcState
//   SODG11_SSCC610_2403701_PLC/SODG11_SSCC610_2403701_PLC Instance <-> EtherCAT Master (EtherCAT)/SS01.N01 (EP9128-0021)/Fix101.N02 (EP1008-0002)
//     Standard Inputs/Fix101.N02/I <-> Channel 1/Input
//     Standard Inputs/Fix101.N02/I @bit 1 <-> Channel 2/Input
//     Standard Inputs/Fix101.N02/I @bit 2 <-> Channel 3/Input
//     Standard Inputs/Fix101.N02/I @bit 3 <-> Channel 4/Input
//     Standard Inputs/Fix101.N02/I @bit 4 <-> Channel 5/Input
//     Standard Inputs/Fix101.N02/I @bit 5 <-> Channel 6/Input
//     Standard Inputs/Fix101.N02/I @bit 6 <-> Channel 7/Input
//     Standard Inputs/Fix101.N02/I @bit 7 <-> Channel 8/Input
//     Standard Inputs/Fix101.N02/InfoData/State <-> InfoData/State
//     Standard Inputs/Fix101.N02/Wc_State <-> WcState/WcState
//   SODG11_SSCC610_2403701_PLC/SODG11_SSCC610_2403701_PLC Instance <-> EtherCAT Master (EtherCAT)/SS01.N01 (EP9128-0021)/Fix101.N03 (EP1008-0002)
//     Standard Inputs/Fix101.N03/I <-> Channel 1/Input
//     Standard Inputs/Fix101.N03/I @bit 1 <-> Channel 2/Input
//     Standard Inputs/Fix101.N03/I @bit 2 <-> Channel 3/Input
//     Standard Inputs/Fix101.N03/I @bit 3 <-> Channel 4/Input
//     Standard Inputs/Fix101.N03/I @bit 4 <-> Channel 5/Input
//     Standard Inputs/Fix101.N03/I @bit 5 <-> Channel 6/Input
//     Standard Inputs/Fix101.N03/I @bit 6 <-> Channel 7/Input
//     Standard Inputs/Fix101.N03/I @bit 7 <-> Channel 8/Input
//     Standard Inputs/Fix101.N03/InfoData/State <-> InfoData/State
//     Standard Inputs/Fix101.N03/Wc_State <-> WcState/WcState
//   SODG11_SSCC610_2403701_PLC/SODG11_SSCC610_2403701_PLC Instance <-> EtherCAT Master (EtherCAT)/SS01.N01 (EP9128-0021)/Fix101.N04 (EP1008-0002)
//     Standard Inputs/Fix101.N04/I <-> Channel 1/Input
//     Standard Inputs/Fix101.N04/I @bit 1 <-> Channel 2/Input
//     Standard Inputs/Fix101.N04/I @bit 2 <-> Channel 3/Input
//     Standard Inputs/Fix101.N04/I @bit 3 <-> Channel 4/Input
//     Standard Inputs/Fix101.N04/I @bit 4 <-> Channel 5/Input
//     Standard Inputs/Fix101.N04/I @bit 5 <-> Channel 6/Input
//     Standard Inputs/Fix101.N04/I @bit 6 <-> Channel 7/Input
//     Standard Inputs/Fix101.N04/I @bit 7 <-> Channel 8/Input
//     Standard Inputs/Fix101.N04/InfoData/State <-> InfoData/State
//     Standard Inputs/Fix101.N04/Wc_State <-> WcState/WcState
//   SODG11_SSCC610_2403701_PLC/SODG11_SSCC610_2403701_PLC Instance <-> EtherCAT Master (EtherCAT)/SS01.N01 (EP9128-0021)/Fix101.N100 (EX260-SEC1)
//     Standard Inputs/Fix101.N100_STAT/InfoData/State <-> InfoData/State
//     Standard Outputs/Fix101.N100/Q <-> Byte 0/Output
//     Standard Outputs/Fix101.N100/Q @bit 8 <-> Byte 1/Output
//     Standard Outputs/Fix101.N100/Q @bit 16 <-> Byte 2/Output
//     Standard Outputs/Fix101.N100/Q @bit 24 <-> Byte 3/Output
//   SODG11_SSCC610_2403701_PLC/SODG11_SSCC610_2403701_PLC Instance <-> EtherCAT Master (EtherCAT)/SS01.N01 (EP9128-0021)/Term 299 (EP9128-1021)
//     Standard Inputs/MAIN.IS01.N01/InfoDataB/State <-> InfoData/State
//     Standard Inputs/MAIN.SS01.N01/InfoDataB/State <-> InfoData/State
//   SODG11_SSCC610_2403701_PLC/SODG11_SSCC610_2403701_PLC Instance <-> EtherCAT Master (EtherCAT)/SS01.N01 (EP9128-0021)/Term 299 (EP9128-1021)/Fix103.N01 (EP1008-0002)
//     Standard Inputs/Fix103.N01/I <-> Channel 1/Input
//     Standard Inputs/Fix103.N01/I @bit 1 <-> Channel 2/Input
//     Standard Inputs/Fix103.N01/I @bit 2 <-> Channel 3/Input
//     Standard Inputs/Fix103.N01/I @bit 3 <-> Channel 4/Input
//     Standard Inputs/Fix103.N01/I @bit 4 <-> Channel 5/Input
//     Standard Inputs/Fix103.N01/I @bit 5 <-> Channel 6/Input
//     Standard Inputs/Fix103.N01/I @bit 6 <-> Channel 7/Input
//     Standard Inputs/Fix103.N01/I @bit 7 <-> Channel 8/Input
//     Standard Inputs/Fix103.N01/InfoData/State <-> InfoData/State
//     Standard Inputs/Fix103.N01/Wc_State <-> WcState/WcState
//   SODG11_SSCC610_2403701_PLC/SODG11_SSCC610_2403701_PLC Instance <-> EtherCAT Master (EtherCAT)/SS01.N01 (EP9128-0021)/Term 299 (EP9128-1021)/Fix103.N02 (EP1008-0002)
//     Standard Inputs/Fix103.N02/I <-> Channel 1/Input
//     Standard Inputs/Fix103.N02/I @bit 1 <-> Channel 2/Input
//     Standard Inputs/Fix103.N02/I @bit 2 <-> Channel 3/Input
//     Standard Inputs/Fix103.N02/I @bit 3 <-> Channel 4/Input
//     Standard Inputs/Fix103.N02/I @bit 4 <-> Channel 5/Input
//     Standard Inputs/Fix103.N02/I @bit 5 <-> Channel 6/Input
//     Standard Inputs/Fix103.N02/I @bit 6 <-> Channel 7/Input
//     Standard Inputs/Fix103.N02/I @bit 7 <-> Channel 8/Input
//     Standard Inputs/Fix103.N02/InfoData/State <-> InfoData/State
//     Standard Inputs/Fix103.N02/Wc_State <-> WcState/WcState
//   SODG11_SSCC610_2403701_PLC/SODG11_SSCC610_2403701_PLC Instance <-> EtherCAT Master (EtherCAT)/SS01.N01 (EP9128-0021)/Term 299 (EP9128-1021)/Fix104.N01 (EP1008-0002)
//     Standard Inputs/Fix104.N01/I <-> Channel 1/Input
//     Standard Inputs/Fix104.N01/I @bit 1 <-> Channel 2/Input
//     Standard Inputs/Fix104.N01/I @bit 2 <-> Channel 3/Input
//     Standard Inputs/Fix104.N01/I @bit 3 <-> Channel 4/Input
//     Standard Inputs/Fix104.N01/I @bit 4 <-> Channel 5/Input
//     Standard Inputs/Fix104.N01/I @bit 5 <-> Channel 6/Input
//     Standard Inputs/Fix104.N01/I @bit 6 <-> Channel 7/Input
//     Standard Inputs/Fix104.N01/I @bit 7 <-> Channel 8/Input
//     Standard Inputs/Fix104.N01/InfoData/State <-> InfoData/State
//     Standard Inputs/Fix104.N01/Wc_State <-> WcState/WcState
//   SODG11_SSCC610_2403701_PLC/SODG11_SSCC610_2403701_PLC Instance <-> EtherCAT Master (EtherCAT)/SS01.N01 (EP9128-0021)/Term 299 (EP9128-1021)/Fix104.N02 (EP1008-0002)
//     Standard Inputs/Fix104.N02/I <-> Channel 1/Input
//     Standard Inputs/Fix104.N02/I @bit 1 <-> Channel 2/Input
//     Standard Inputs/Fix104.N02/I @bit 2 <-> Channel 3/Input
//     Standard Inputs/Fix104.N02/I @bit 3 <-> Channel 4/Input
//     Standard Inputs/Fix104.N02/I @bit 4 <-> Channel 5/Input
//     Standard Inputs/Fix104.N02/I @bit 5 <-> Channel 6/Input
//     Standard Inputs/Fix104.N02/I @bit 6 <-> Channel 7/Input
//     Standard Inputs/Fix104.N02/I @bit 7 <-> Channel 8/Input
//     Standard Inputs/Fix104.N02/InfoData/State <-> InfoData/State
//     Standard Inputs/Fix104.N02/Wc_State <-> WcState/WcState
//   SODG11_SSCC610_2403701_PLC/SODG11_SSCC610_2403701_PLC Instance <-> EtherCAT Master (EtherCAT)/SS01.N01 (EP9128-0021)/Term 299 (EP9128-1021)/Fix105.N01 (EP1008-0002)
//     Standard Inputs/Fix105.N01/I <-> Channel 1/Input
//     Standard Inputs/Fix105.N01/I @bit 1 <-> Channel 2/Input
//     Standard Inputs/Fix105.N01/I @bit 2 <-> Channel 3/Input
//     Standard Inputs/Fix105.N01/I @bit 3 <-> Channel 4/Input
//     Standard Inputs/Fix105.N01/I @bit 4 <-> Channel 5/Input
//     Standard Inputs/Fix105.N01/I @bit 5 <-> Channel 6/Input
//     Standard Inputs/Fix105.N01/I @bit 6 <-> Channel 7/Input
//     Standard Inputs/Fix105.N01/I @bit 7 <-> Channel 8/Input
//     Standard Inputs/Fix105.N01/InfoData/State <-> InfoData/State
//     Standard Inputs/Fix105.N01/Wc_State <-> WcState/WcState
//   SODG11_SSCC610_2403701_PLC/SODG11_SSCC610_2403701_PLC Instance <-> EtherCAT Master (EtherCAT)/SS01.N01 (EP9128-0021)/Term 299 (EP9128-1021)/Fix105.N02 (EP1008-0002)
//     Standard Inputs/Fix105.N02/I <-> Channel 1/Input
//     Standard Inputs/Fix105.N02/I @bit 1 <-> Channel 2/Input
//     Standard Inputs/Fix105.N02/I @bit 2 <-> Channel 3/Input
//     Standard Inputs/Fix105.N02/I @bit 3 <-> Channel 4/Input
//     Standard Inputs/Fix105.N02/I @bit 4 <-> Channel 5/Input
//     Standard Inputs/Fix105.N02/I @bit 5 <-> Channel 6/Input
//     Standard Inputs/Fix105.N02/I @bit 6 <-> Channel 7/Input
//     Standard Inputs/Fix105.N02/I @bit 7 <-> Channel 8/Input
//     Standard Inputs/Fix105.N02/InfoData/State <-> InfoData/State
//     Standard Inputs/Fix105.N02/Wc_State <-> WcState/WcState
//   SODG11_SSCC610_2403701_PLC/SODG11_SSCC610_2403701_PLC Instance <-> EtherCAT Master (EtherCAT)/SS01.N01 (EP9128-0021)/Term 299 (EP9128-1021)/VFD01 (ATV320 EtherCAT)
//     Standard Inputs/MAIN.VFD01.Status_Word <-> Inputs/Status word
//     Standard Inputs/MAIN.VFD01.VFD_State/InfoData/State <-> InfoData/State
//     Standard Outputs/MAIN.VFD01.Control_Word <-> Outputs/Control word
//     Standard Outputs/MAIN.VFD01.Target_Velocity <-> Outputs/Target Velocity
//   SODG11_SSCC610_2403701_PLC/SODG11_SSCC610_2403701_PLC Instance <-> EtherCAT Master (EtherCAT)/SS01.N01 (EP9128-0021)/Term 299 (EP9128-1021)/VFD02 (ATV320 EtherCAT)
//     Standard Inputs/MAIN.VFD02.Status_Word <-> Inputs/Status word
//     Standard Inputs/MAIN.VFD02.VFD_State/InfoData/State <-> InfoData/State
//     Standard Outputs/MAIN.VFD02.Control_Word <-> Outputs/Control word
//     Standard Outputs/MAIN.VFD02.Target_Velocity <-> Outputs/Target Velocity
//   SODG11_SSCC610_2403701_PLC/SODG11_SSCC610_2403701_PLC Instance <-> EtherCAT Master (EtherCAT)/SS01.N01 (EP9128-0021)/Term 301 (EP9128-2021)
//     Standard Inputs/MAIN.IS01.N01/InfoDataC/State <-> InfoData/State
//     Standard Inputs/MAIN.SS01.N01/InfoDataC/State <-> InfoData/State
//   SODG11_SSCC610_2403701_PLC/SODG11_SSCC610_2403701_PLC Instance <-> EtherCAT Master (EtherCAT)/SS01.N01 (EP9128-0021)/VertiGuard.N01 (EP2028-0002)
//     Standard Inputs/MAIN.VertiGuard_N01_STAT/InfoData/State <-> InfoData/State
//     Standard Outputs/MAIN.VertiGuard_N01/Q <-> Channel 1/Output
//     Standard Outputs/MAIN.VertiGuard_N01/Q @bit 1 <-> Channel 2/Output
//     Standard Outputs/MAIN.VertiGuard_N01/Q @bit 2 <-> Channel 3/Output
//     Standard Outputs/MAIN.VertiGuard_N01/Q @bit 3 <-> Channel 4/Output
//     Standard Outputs/MAIN.VertiGuard_N01/Q @bit 4 <-> Channel 5/Output
//     Standard Outputs/MAIN.VertiGuard_N01/Q @bit 5 <-> Channel 6/Output
//     Standard Outputs/MAIN.VertiGuard_N01/Q @bit 6 <-> Channel 7/Output
//     Standard Outputs/MAIN.VertiGuard_N01/Q @bit 7 <-> Channel 8/Output
//   SODG11_SSCC610_2403701_PLC/SODG11_SSCC610_2403701_PLC Instance <-> EtherCAT Master (EtherCAT)/SS01.N01 (EP9128-0021)/VertiGuard.N02 (EP1908)
//     Standard Inputs/MAIN.VertiGuard_N02/I <-> Module 1 (FSOE)/FSOE Inputs/FSOE/InputChannel1
//     Standard Inputs/MAIN.VertiGuard_N02/I @bit 1 <-> Module 1 (FSOE)/FSOE Inputs/FSOE/InputChannel2
//     Standard Inputs/MAIN.VertiGuard_N02/I @bit 2 <-> Module 1 (FSOE)/FSOE Inputs/FSOE/InputChannel3
//     Standard Inputs/MAIN.VertiGuard_N02/I @bit 3 <-> Module 1 (FSOE)/FSOE Inputs/FSOE/InputChannel4
//     Standard Inputs/MAIN.VertiGuard_N02/I @bit 4 <-> Module 1 (FSOE)/FSOE Inputs/FSOE/InputChannel5
//     Standard Inputs/MAIN.VertiGuard_N02/I @bit 5 <-> Module 1 (FSOE)/FSOE Inputs/FSOE/InputChannel6
//     Standard Inputs/MAIN.VertiGuard_N02/I @bit 6 <-> Module 1 (FSOE)/FSOE Inputs/FSOE/InputChannel7
//     Standard Inputs/MAIN.VertiGuard_N02/I @bit 7 <-> Module 1 (FSOE)/FSOE Inputs/FSOE/InputChannel8
//     Standard Inputs/MAIN.VertiGuard_N02/InfoData/State <-> InfoData/State
//   SODG11_SSCC610_2403701_PLC/SODG11_SSCC610_2403701_PLC Instance <-> EtherCAT Master (EtherCAT)/SS01.N02 (EP1008-0002)
//     Standard Inputs/MAIN.SS01.N02/I <-> Channel 1/Input
//     Standard Inputs/MAIN.SS01.N02/I @bit 1 <-> Channel 2/Input
//     Standard Inputs/MAIN.SS01.N02/I @bit 2 <-> Channel 3/Input
//     Standard Inputs/MAIN.SS01.N02/I @bit 3 <-> Channel 4/Input
//     Standard Inputs/MAIN.SS01.N02/I @bit 4 <-> Channel 5/Input
//     Standard Inputs/MAIN.SS01.N02/I @bit 5 <-> Channel 6/Input
//     Standard Inputs/MAIN.SS01.N02/I @bit 6 <-> Channel 7/Input
//     Standard Inputs/MAIN.SS01.N02/I @bit 7 <-> Channel 8/Input
//     Standard Inputs/MAIN.SS01.N02/InfoData/State <-> InfoData/State
//     Standard Inputs/MAIN.SS01.N02/Wc_State <-> WcState/WcState
//   SODG11_SSCC610_2403701_PLC/SODG11_SSCC610_2403701_PLC Instance <-> EtherCAT Master (EtherCAT)/SS01.N03 (EP2028-0002)
//     Standard Inputs/MAIN.SS01.N03_STAT/InfoData/State <-> InfoData/State
//     Standard Outputs/MAIN.SS01.N03/Q <-> Channel 1/Output
//     Standard Outputs/MAIN.SS01.N03/Q @bit 1 <-> Channel 2/Output
//     Standard Outputs/MAIN.SS01.N03/Q @bit 2 <-> Channel 3/Output
//     Standard Outputs/MAIN.SS01.N03/Q @bit 3 <-> Channel 4/Output
//     Standard Outputs/MAIN.SS01.N03/Q @bit 4 <-> Channel 5/Output
//     Standard Outputs/MAIN.SS01.N03/Q @bit 5 <-> Channel 6/Output
//     Standard Outputs/MAIN.SS01.N03/Q @bit 6 <-> Channel 7/Output
//     Standard Outputs/MAIN.SS01.N03/Q @bit 7 <-> Channel 8/Output
//   SODG11_SSCC610_2403701_PLC/SODG11_SSCC610_2403701_PLC Instance <-> EtherCAT Master (EtherCAT)/SS01.N04 (EP9214-0023)
//     Standard Inputs/MAIN.SS01.N04_STAT/Channel_1/Channel_Error <-> DPO Inputs Channel 1/Channel Error
//     Standard Inputs/MAIN.SS01.N04_STAT/Channel_2/Channel_Error <-> DPO Inputs Channel 2/Channel Error
//     Standard Inputs/MAIN.SS01.N04_STAT/Channel_3/Channel_Error <-> DPO Inputs Channel 3/Channel Error
//     Standard Inputs/MAIN.SS01.N04_STAT/Channel_4/Channel_Error <-> DPO Inputs Channel 4/Channel Error
//     Standard Inputs/MAIN.SS01.N04_STAT/Channel_1/Error_Up <-> DPO Inputs Channel 1/Error Up
//     Standard Inputs/MAIN.SS01.N04_STAT/Channel_2/Error_Up <-> DPO Inputs Channel 2/Error Up
//     Standard Inputs/MAIN.SS01.N04_STAT/Channel_3/Error_Up <-> DPO Inputs Channel 3/Error Up
//     Standard Inputs/MAIN.SS01.N04_STAT/Channel_4/Error_Up <-> DPO Inputs Channel 4/Error Up
//     Standard Inputs/MAIN.SS01.N04_STAT/Channel_1/Error_Us <-> DPO Inputs Channel 1/Error Us
//     Standard Inputs/MAIN.SS01.N04_STAT/Channel_2/Error_Us <-> DPO Inputs Channel 2/Error Us
//     Standard Inputs/MAIN.SS01.N04_STAT/Channel_3/Error_Us <-> DPO Inputs Channel 3/Error Us
//     Standard Inputs/MAIN.SS01.N04_STAT/Channel_4/Error_Us <-> DPO Inputs Channel 4/Error Us
//     Standard Inputs/MAIN.SS01.N04_STAT/Channel_1/Status_Up <-> DPO Inputs Channel 1/Status Up
//     Standard Inputs/MAIN.SS01.N04_STAT/Channel_2/Status_Up <-> DPO Inputs Channel 2/Status Up
//     Standard Inputs/MAIN.SS01.N04_STAT/Channel_3/Status_Up <-> DPO Inputs Channel 3/Status Up
//     Standard Inputs/MAIN.SS01.N04_STAT/Channel_4/Status_Up <-> DPO Inputs Channel 4/Status Up
//     Standard Inputs/MAIN.SS01.N04_STAT/Channel_1/Status_Us <-> DPO Inputs Channel 1/Status Us
//     Standard Inputs/MAIN.SS01.N04_STAT/Channel_2/Status_Us <-> DPO Inputs Channel 2/Status Us
//     Standard Inputs/MAIN.SS01.N04_STAT/Channel_3/Status_Us <-> DPO Inputs Channel 3/Status Us
//     Standard Inputs/MAIN.SS01.N04_STAT/Channel_4/Status_Us <-> DPO Inputs Channel 4/Status Us
//     Standard Inputs/MAIN.SS01.N04_STAT/Channel_1/SyncError <-> DPO Inputs Channel 1/Sync error
//     Standard Inputs/MAIN.SS01.N04_STAT/Channel_2/SyncError <-> DPO Inputs Channel 2/Sync error
//     Standard Inputs/MAIN.SS01.N04_STAT/Channel_3/SyncError <-> DPO Inputs Channel 3/Sync error
//     Standard Inputs/MAIN.SS01.N04_STAT/Channel_4/SyncError <-> DPO Inputs Channel 4/Sync error
//     Standard Inputs/MAIN.SS01.N04_STAT/Channel_1/TxPDO_State <-> DPO Inputs Channel 1/TxPDO State
//     Standard Inputs/MAIN.SS01.N04_STAT/Channel_2/TxPDO_State <-> DPO Inputs Channel 2/TxPDO State
//     Standard Inputs/MAIN.SS01.N04_STAT/Channel_3/TxPDO_State <-> DPO Inputs Channel 3/TxPDO State
//     Standard Inputs/MAIN.SS01.N04_STAT/Channel_4/TxPDO_State <-> DPO Inputs Channel 4/TxPDO State
//     Standard Inputs/MAIN.SS01.N04_STAT/Channel_1/TxPDO_Toggle <-> DPO Inputs Channel 1/TxPDO Toggle
//     Standard Inputs/MAIN.SS01.N04_STAT/Channel_2/TxPDO_Toggle <-> DPO Inputs Channel 2/TxPDO Toggle
//     Standard Inputs/MAIN.SS01.N04_STAT/Channel_3/TxPDO_Toggle <-> DPO Inputs Channel 3/TxPDO Toggle
//     Standard Inputs/MAIN.SS01.N04_STAT/Channel_4/TxPDO_Toggle <-> DPO Inputs Channel 4/TxPDO Toggle
//     Standard Inputs/MAIN.SS01.N04_STAT/Channel_1/Warning_Up <-> DPO Inputs Channel 1/Warning Up
//     Standard Inputs/MAIN.SS01.N04_STAT/Channel_2/Warning_Up <-> DPO Inputs Channel 2/Warning Up
//     Standard Inputs/MAIN.SS01.N04_STAT/Channel_3/Warning_Up <-> DPO Inputs Channel 3/Warning Up
//     Standard Inputs/MAIN.SS01.N04_STAT/Channel_4/Warning_Up <-> DPO Inputs Channel 4/Warning Up
//     Standard Inputs/MAIN.SS01.N04_STAT/Channel_1/Warning_Us <-> DPO Inputs Channel 1/Warning Us
//     Standard Inputs/MAIN.SS01.N04_STAT/Channel_2/Warning_Us <-> DPO Inputs Channel 2/Warning Us
//     Standard Inputs/MAIN.SS01.N04_STAT/Channel_3/Warning_Us <-> DPO Inputs Channel 3/Warning Us
//     Standard Inputs/MAIN.SS01.N04_STAT/Channel_4/Warning_Us <-> DPO Inputs Channel 4/Warning Us
//     Standard Inputs/MAIN.SS01.N04_STAT/Device/Global_Error_Bit <-> DPO Inputs Device/Global Error Bit
//     Standard Inputs/MAIN.SS01.N04_STAT/Device/Reset_Input <-> DPO Inputs Device/Reset Input
//     Standard Inputs/MAIN.SS01.N04_STAT/Device/Temperature_Error <-> DPO Inputs Device/Temperature Error
//     Standard Inputs/MAIN.SS01.N04_STAT/Device/Temperature_Warning <-> DPO Inputs Device/Temperature Warning
//     Standard Inputs/MAIN.SS01.N04_STAT/Device/TxPDO_State <-> DPO Inputs Device/TxPDO State
//     Standard Inputs/MAIN.SS01.N04_STAT/Device/TxPDO_Toggle <-> DPO Inputs Device/TxPDO Toggle
//     Standard Inputs/MAIN.SS01.N04_STAT/Device/Up_Error <-> DPO Inputs Device/Up Error
//     Standard Inputs/MAIN.SS01.N04_STAT/Device/Up_Warning <-> DPO Inputs Device/Up Warning
//     Standard Inputs/MAIN.SS01.N04_STAT/Device/Us_Error <-> DPO Inputs Device/Us Error
//     Standard Inputs/MAIN.SS01.N04_STAT/Device/Us_Warning <-> DPO Inputs Device/Us Warning
//     Standard Inputs/MAIN.SS01.N04_STAT/InfoData/AdsAddr/netId <-> InfoData/AdsAddr/netId
//     Standard Inputs/MAIN.SS01.N04_STAT/InfoData/AdsAddr/port <-> InfoData/AdsAddr/port
//     Standard Inputs/MAIN.SS01.N04_STAT/InfoData/State <-> InfoData/State
//     Standard Inputs/MAIN.SS01.N04_STAT/Wc_State <-> WcState/WcState
//     Standard Outputs/MAIN.SS01.N04_CMD/Channel1/Output_Up <-> DPO Outputs Channel 1/Output Up
//     Standard Outputs/MAIN.SS01.N04_CMD/Channel2/Output_Up <-> DPO Outputs Channel 2/Output Up
//     Standard Outputs/MAIN.SS01.N04_CMD/Channel3/Output_Up <-> DPO Outputs Channel 3/Output Up
//     Standard Outputs/MAIN.SS01.N04_CMD/Channel4/Output_Up <-> DPO Outputs Channel 4/Output Up
//     Standard Outputs/MAIN.SS01.N04_CMD/Channel1/Output_Us <-> DPO Outputs Channel 1/Output Us
//     Standard Outputs/MAIN.SS01.N04_CMD/Channel2/Output_Us <-> DPO Outputs Channel 2/Output Us
//     Standard Outputs/MAIN.SS01.N04_CMD/Channel3/Output_Us <-> DPO Outputs Channel 3/Output Us
//     Standard Outputs/MAIN.SS01.N04_CMD/Channel4/Output_Us <-> DPO Outputs Channel 4/Output Us
//     Standard Outputs/MAIN.SS01.N04_CMD/Channel1/Reset_Up <-> DPO Outputs Channel 1/Reset Up
//     Standard Outputs/MAIN.SS01.N04_CMD/Channel2/Reset_Up <-> DPO Outputs Channel 2/Reset Up
//     Standard Outputs/MAIN.SS01.N04_CMD/Channel3/Reset_Up <-> DPO Outputs Channel 3/Reset Up
//     Standard Outputs/MAIN.SS01.N04_CMD/Channel4/Reset_Up <-> DPO Outputs Channel 4/Reset Up
//     Standard Outputs/MAIN.SS01.N04_CMD/Channel1/Reset_Us <-> DPO Outputs Channel 1/Reset Us
//     Standard Outputs/MAIN.SS01.N04_CMD/Channel2/Reset_Us <-> DPO Outputs Channel 2/Reset Us
//     Standard Outputs/MAIN.SS01.N04_CMD/Channel3/Reset_Us <-> DPO Outputs Channel 3/Reset Us
//     Standard Outputs/MAIN.SS01.N04_CMD/Channel4/Reset_Us <-> DPO Outputs Channel 4/Reset Us
//     Standard Outputs/MAIN.SS01.N04_CMD/Device/Enable_Control_Via_Fieldbus <-> DPO Outputs Device/Enable Control Via Fieldbus
//     Standard Outputs/MAIN.SS01.N04_CMD/Device/Global_Reset <-> DPO Outputs Device/Global Reset
//   SODG11_SSCC610_2403701_PLC/SODG11_SSCC610_2403701_PLC Instance <-> PD01.T05 (EL6731)/SIC01.N10 (GSD Box) (UNIGATE IC - Profibus)
//     Standard Inputs/MAIN.SIC01.SICMarker_Inputs/Input0_0 <-> Module 1 (E10-240 bytes I/O)/Inputs/E10-240 bytes I/O_0_0
//     Standard Inputs/MAIN.SIC01.SICMarker_Inputs/Input0_1 <-> Module 1 (E10-240 bytes I/O)/Inputs/E10-240 bytes I/O_0_1
//     Standard Inputs/MAIN.SIC01.SICMarker_Inputs/Input0_10 <-> Module 1 (E10-240 bytes I/O)/Inputs/E10-240 bytes I/O_0_10
//     Standard Inputs/MAIN.SIC01.SICMarker_Inputs/Input0_11 <-> Module 1 (E10-240 bytes I/O)/Inputs/E10-240 bytes I/O_0_11
//     Standard Inputs/MAIN.SIC01.SICMarker_Inputs/Input0_12 <-> Module 1 (E10-240 bytes I/O)/Inputs/E10-240 bytes I/O_0_12
//     Standard Inputs/MAIN.SIC01.SICMarker_Inputs/Input0_13 <-> Module 1 (E10-240 bytes I/O)/Inputs/E10-240 bytes I/O_0_13
//     Standard Inputs/MAIN.SIC01.SICMarker_Inputs/Input0_14 <-> Module 1 (E10-240 bytes I/O)/Inputs/E10-240 bytes I/O_0_14
//     Standard Inputs/MAIN.SIC01.SICMarker_Inputs/Input0_2 <-> Module 1 (E10-240 bytes I/O)/Inputs/E10-240 bytes I/O_0_2
//     Standard Inputs/MAIN.SIC01.SICMarker_Inputs/Input0_3 <-> Module 1 (E10-240 bytes I/O)/Inputs/E10-240 bytes I/O_0_3
//     Standard Inputs/MAIN.SIC01.SICMarker_Inputs/Input0_4 <-> Module 1 (E10-240 bytes I/O)/Inputs/E10-240 bytes I/O_0_4
//     Standard Inputs/MAIN.SIC01.SICMarker_Inputs/Input0_5 <-> Module 1 (E10-240 bytes I/O)/Inputs/E10-240 bytes I/O_0_5
//     Standard Inputs/MAIN.SIC01.SICMarker_Inputs/Input0_6 <-> Module 1 (E10-240 bytes I/O)/Inputs/E10-240 bytes I/O_0_6
//     Standard Inputs/MAIN.SIC01.SICMarker_Inputs/Input0_7 <-> Module 1 (E10-240 bytes I/O)/Inputs/E10-240 bytes I/O_0_7
//     Standard Inputs/MAIN.SIC01.SICMarker_Inputs/Input0_8 <-> Module 1 (E10-240 bytes I/O)/Inputs/E10-240 bytes I/O_0_8
//     Standard Inputs/MAIN.SIC01.SICMarker_Inputs/Input0_9 <-> Module 1 (E10-240 bytes I/O)/Inputs/E10-240 bytes I/O_0_9
//     Standard Inputs/MAIN.SIC01.SICMarker_Inputs/Inputs/DpState <-> Inputs/DpState
//     Standard Inputs/MAIN.SIC01.SICMarker_Inputs/Inputs/ExtDiagFlag <-> Inputs/ExtDiagFlag
//     Standard Outputs/MAIN.SIC01.SICMarker_Outputs/Output1_0 <-> Module 1 (E10-240 bytes I/O)/Outputs/E10-240 bytes I/O_1_0
//     Standard Outputs/MAIN.SIC01.SICMarker_Outputs/Output1_1 <-> Module 1 (E10-240 bytes I/O)/Outputs/E10-240 bytes I/O_1_1
//     Standard Outputs/MAIN.SIC01.SICMarker_Outputs/Output1_10 <-> Module 1 (E10-240 bytes I/O)/Outputs/E10-240 bytes I/O_1_10
//     Standard Outputs/MAIN.SIC01.SICMarker_Outputs/Output1_11 <-> Module 1 (E10-240 bytes I/O)/Outputs/E10-240 bytes I/O_1_11
//     Standard Outputs/MAIN.SIC01.SICMarker_Outputs/Output1_12 <-> Module 1 (E10-240 bytes I/O)/Outputs/E10-240 bytes I/O_1_12
//     Standard Outputs/MAIN.SIC01.SICMarker_Outputs/Output1_13 <-> Module 1 (E10-240 bytes I/O)/Outputs/E10-240 bytes I/O_1_13
//     Standard Outputs/MAIN.SIC01.SICMarker_Outputs/Output1_14 <-> Module 1 (E10-240 bytes I/O)/Outputs/E10-240 bytes I/O_1_14
//     Standard Outputs/MAIN.SIC01.SICMarker_Outputs/Output1_2 <-> Module 1 (E10-240 bytes I/O)/Outputs/E10-240 bytes I/O_1_2
//     Standard Outputs/MAIN.SIC01.SICMarker_Outputs/Output1_3 <-> Module 1 (E10-240 bytes I/O)/Outputs/E10-240 bytes I/O_1_3
//     Standard Outputs/MAIN.SIC01.SICMarker_Outputs/Output1_4 <-> Module 1 (E10-240 bytes I/O)/Outputs/E10-240 bytes I/O_1_4
//     Standard Outputs/MAIN.SIC01.SICMarker_Outputs/Output1_5 <-> Module 1 (E10-240 bytes I/O)/Outputs/E10-240 bytes I/O_1_5
//     Standard Outputs/MAIN.SIC01.SICMarker_Outputs/Output1_6 <-> Module 1 (E10-240 bytes I/O)/Outputs/E10-240 bytes I/O_1_6
//     Standard Outputs/MAIN.SIC01.SICMarker_Outputs/Output1_7 <-> Module 1 (E10-240 bytes I/O)/Outputs/E10-240 bytes I/O_1_7
//     Standard Outputs/MAIN.SIC01.SICMarker_Outputs/Output1_8 <-> Module 1 (E10-240 bytes I/O)/Outputs/E10-240 bytes I/O_1_8
//     Standard Outputs/MAIN.SIC01.SICMarker_Outputs/Output1_9 <-> Module 1 (E10-240 bytes I/O)/Outputs/E10-240 bytes I/O_1_9
//   SODG11_SSCC610_2403701_PLC/SODG11_SSCC610_2403701_PLC Instance <-> PD01.T05 (EL6731)/SIC01.N20 (GSD Box) (UNIGATE IC - Profibus)
//     Standard Inputs/MAIN.SIC02.SICMarker_Inputs/Input0_0 <-> Module 1 (E10-240 bytes I/O)/Inputs/E10-240 bytes I/O_0_0
//     Standard Inputs/MAIN.SIC02.SICMarker_Inputs/Input0_1 <-> Module 1 (E10-240 bytes I/O)/Inputs/E10-240 bytes I/O_0_1
//     Standard Inputs/MAIN.SIC02.SICMarker_Inputs/Input0_10 <-> Module 1 (E10-240 bytes I/O)/Inputs/E10-240 bytes I/O_0_10
//     Standard Inputs/MAIN.SIC02.SICMarker_Inputs/Input0_11 <-> Module 1 (E10-240 bytes I/O)/Inputs/E10-240 bytes I/O_0_11
//     Standard Inputs/MAIN.SIC02.SICMarker_Inputs/Input0_12 <-> Module 1 (E10-240 bytes I/O)/Inputs/E10-240 bytes I/O_0_12
//     Standard Inputs/MAIN.SIC02.SICMarker_Inputs/Input0_13 <-> Module 1 (E10-240 bytes I/O)/Inputs/E10-240 bytes I/O_0_13
//     Standard Inputs/MAIN.SIC02.SICMarker_Inputs/Input0_14 <-> Module 1 (E10-240 bytes I/O)/Inputs/E10-240 bytes I/O_0_14
//     Standard Inputs/MAIN.SIC02.SICMarker_Inputs/Input0_2 <-> Module 1 (E10-240 bytes I/O)/Inputs/E10-240 bytes I/O_0_2
//     Standard Inputs/MAIN.SIC02.SICMarker_Inputs/Input0_3 <-> Module 1 (E10-240 bytes I/O)/Inputs/E10-240 bytes I/O_0_3
//     Standard Inputs/MAIN.SIC02.SICMarker_Inputs/Input0_4 <-> Module 1 (E10-240 bytes I/O)/Inputs/E10-240 bytes I/O_0_4
//     Standard Inputs/MAIN.SIC02.SICMarker_Inputs/Input0_5 <-> Module 1 (E10-240 bytes I/O)/Inputs/E10-240 bytes I/O_0_5
//     Standard Inputs/MAIN.SIC02.SICMarker_Inputs/Input0_6 <-> Module 1 (E10-240 bytes I/O)/Inputs/E10-240 bytes I/O_0_6
//     Standard Inputs/MAIN.SIC02.SICMarker_Inputs/Input0_7 <-> Module 1 (E10-240 bytes I/O)/Inputs/E10-240 bytes I/O_0_7
//     Standard Inputs/MAIN.SIC02.SICMarker_Inputs/Input0_8 <-> Module 1 (E10-240 bytes I/O)/Inputs/E10-240 bytes I/O_0_8
//     Standard Inputs/MAIN.SIC02.SICMarker_Inputs/Input0_9 <-> Module 1 (E10-240 bytes I/O)/Inputs/E10-240 bytes I/O_0_9
//     Standard Inputs/MAIN.SIC02.SICMarker_Inputs/Inputs/DpState <-> Inputs/DpState
//     Standard Inputs/MAIN.SIC02.SICMarker_Inputs/Inputs/ExtDiagFlag <-> Inputs/ExtDiagFlag
//     Standard Outputs/MAIN.SIC02.SICMarker_Outputs/Output1_0 <-> Module 1 (E10-240 bytes I/O)/Outputs/E10-240 bytes I/O_1_0
//     Standard Outputs/MAIN.SIC02.SICMarker_Outputs/Output1_1 <-> Module 1 (E10-240 bytes I/O)/Outputs/E10-240 bytes I/O_1_1
//     Standard Outputs/MAIN.SIC02.SICMarker_Outputs/Output1_10 <-> Module 1 (E10-240 bytes I/O)/Outputs/E10-240 bytes I/O_1_10
//     Standard Outputs/MAIN.SIC02.SICMarker_Outputs/Output1_11 <-> Module 1 (E10-240 bytes I/O)/Outputs/E10-240 bytes I/O_1_11
//     Standard Outputs/MAIN.SIC02.SICMarker_Outputs/Output1_12 <-> Module 1 (E10-240 bytes I/O)/Outputs/E10-240 bytes I/O_1_12
//     Standard Outputs/MAIN.SIC02.SICMarker_Outputs/Output1_13 <-> Module 1 (E10-240 bytes I/O)/Outputs/E10-240 bytes I/O_1_13
//     Standard Outputs/MAIN.SIC02.SICMarker_Outputs/Output1_14 <-> Module 1 (E10-240 bytes I/O)/Outputs/E10-240 bytes I/O_1_14
//     Standard Outputs/MAIN.SIC02.SICMarker_Outputs/Output1_2 <-> Module 1 (E10-240 bytes I/O)/Outputs/E10-240 bytes I/O_1_2
//     Standard Outputs/MAIN.SIC02.SICMarker_Outputs/Output1_3 <-> Module 1 (E10-240 bytes I/O)/Outputs/E10-240 bytes I/O_1_3
//     Standard Outputs/MAIN.SIC02.SICMarker_Outputs/Output1_4 <-> Module 1 (E10-240 bytes I/O)/Outputs/E10-240 bytes I/O_1_4
//     Standard Outputs/MAIN.SIC02.SICMarker_Outputs/Output1_5 <-> Module 1 (E10-240 bytes I/O)/Outputs/E10-240 bytes I/O_1_5
//     Standard Outputs/MAIN.SIC02.SICMarker_Outputs/Output1_6 <-> Module 1 (E10-240 bytes I/O)/Outputs/E10-240 bytes I/O_1_6
//     Standard Outputs/MAIN.SIC02.SICMarker_Outputs/Output1_7 <-> Module 1 (E10-240 bytes I/O)/Outputs/E10-240 bytes I/O_1_7
//     Standard Outputs/MAIN.SIC02.SICMarker_Outputs/Output1_8 <-> Module 1 (E10-240 bytes I/O)/Outputs/E10-240 bytes I/O_1_8
//     Standard Outputs/MAIN.SIC02.SICMarker_Outputs/Output1_9 <-> Module 1 (E10-240 bytes I/O)/Outputs/E10-240 bytes I/O_1_9

CONFIGURATION SODG11_SSCC610_2403701_PLC
    RESOURCE PLC ON TwinCAT3
        TASK Standard(INTERVAL := T#20ms, PRIORITY := 11);
        PROGRAM MAIN WITH Standard : MAIN;
    END_RESOURCE
END_CONFIGURATION

// ---- Data types/ATI/udt_ATI_Input_20150203.TcDUT
(*udt (user defined type) of ATI Input Data:
	auth. Rob Remillard of Sodecia GTAC
	Version 20150203
		- Initial Concept

	Last Edit: Feb 3, 2015, rr
*)
TYPE udt_ATI_Input_20150203 :

	STRUCT

		(*Status Of EtherCat Slave*)
		InfoData: udt_ECATSlave_Status;
		(*Input Bytes*)
		Byte0: BYTE;
		Byte1: BYTE;
		Byte2: BYTE;
		Byte3: BYTE;
		Byte456: UDINT;
		Byte7: BYTE;

	END_STRUCT

END_TYPE

// ---- Data types/ATI/udt_ATI_Output_20150203.TcDUT
(*udt (user defined type) of ATI Output Data:
	auth. Rob Remillard of Sodecia GTAC
	Version 20150203
		- Initial Concept

	Last Edit: Feb 3, 2015, rr
*)
TYPE udt_ATI_Output_20150203 :

	STRUCT

		(*Output Bytes*)
		Byte0: BYTE;
		Byte1: BYTE;
		Byte2: BYTE;
		Byte3: BYTE;
		Byte4: BYTE;
		Byte5: BYTE;
		Byte6: BYTE;
		Byte7: BYTE;

	END_STRUCT

END_TYPE

// ---- Data types/Beckhoff IO udts/udt_AdsAddr.TcDUT
TYPE udt_AdsAddr :
STRUCT
(*Used to read in the ADS address of the AX5805*)
(*Data structure must remain in this order*)
	netId:		ARRAY [0..5] OF USINT;
END_STRUCT
END_TYPE

// ---- Data types/Beckhoff IO udts/udt_AdsAddr_AX5805.TcDUT
TYPE udt_AdsAddr_AX5805 :
STRUCT
(*Used to read in the ADS address of the AX5805*)
(*Data structure must remain in this order*)
	Addr:		udt_AdsAddr;
	port:			UINT;
END_STRUCT
END_TYPE

// ---- Data types/Beckhoff IO udts/udt_CU1128_20180507.TcDUT
(*udt (user defined type) of Beckhoff CU1128 - EtherCAT Junction:
	
------------------------------------------------------------------------
REVISION NOTES:
	Original Author(s): b.lekx-toniolo
	Version 20150812
		- Initial Concept

------------------------------------------------------------------------
*)
TYPE udt_CU1128_20180507 :
STRUCT
	InfoData: udt_ECATSlave_Status_CU1128;
	InfoDataB: udt_ECATSlave_Status_CU1128;
	InfoDataC: udt_ECATSlave_Status_CU1128;
END_STRUCT
END_TYPE

// ---- Data types/Beckhoff IO udts/udt_ECATMaster_InfoData_20121206.TcDUT
(*udt (user defined type) of Infodata Portion of Beckhoff Type EtherCAT Master:
	auth. Brent Lekx-Toniolo of Sodecia GTAC
	Version 20121206
		- Initial Concept

	Last Edit: December 6th, 2012, blt

*)
TYPE udt_ECATMaster_InfoData_20121206 :
	STRUCT
	ChangeCount: UINT;
	DevID: UINT;
	AmsNetId: ARRAY [0..5] OF USINT;
	CfgSlaveCount: UINT;
	END_STRUCT
END_TYPE

// ---- Data types/Beckhoff IO udts/udt_ECATMaster_Status.TcDUT
(*udt (user defined type) of Beckhoff Type EtherCAT Master:
	auth. Brent Lekx-Toniolo of Toniolo Research & Development Inc.; 
	July 2010; version 1.0*)



TYPE udt_ECATMaster_Status :
STRUCT
	Frm0State: UINT;
	(*
	0x0001 = 1. EtherCAT command NOT sent (NOP requested)
	0x0002 = 2. EtherCAT command NOT sent (NOP requested)
	0x0004 = 3. EtherCAT command NOT sent (NOP requested)
	...
	0x4000 = 15. EtherCAT command NOT sent (NOP requested)
	0x8000 = complete frame NOT sent*)
	Frm0WcState: UINT;
	(*
	0x0001 = wrong working counter of 1. EtherCAT command received
	0x0002 = wrong working counter of 2. EtherCAT command received
	0x0004 = wrong working counter of 3. EtherCAT command received
	...
	0x4000 = wrong working counter of 15. EtherCAT command received
	0x8000 = complete frame missing*)
	FR5State: UINT;
	(*
	0x0001 = 1. EtherCAT command NOT sent (NOP requested)
	0x0002 = 2. EtherCAT command NOT sent (NOP requested)
	0x0004 = 3. EtherCAT command NOT sent (NOP requested)
	...
	0x4000 = 15. EtherCAT command NOT sent (NOP requested)
	0x8000 = complete frame NOT sent*)
	FR5WcState: UINT;
	(*
	0x0001 = wrong working counter of 1. EtherCAT command received
	0x0002 = wrong working counter of 2. EtherCAT command received
	0x0004 = wrong working counter of 3. EtherCAT command received
	...
	0x4000 = wrong working counter of 15. EtherCAT command received
	0x8000 = complete frame missing*)
	FR7State: UINT;
	(*
	0x0001 = 1. EtherCAT command NOT sent (NOP requested)
	0x0002 = 2. EtherCAT command NOT sent (NOP requested)
	0x0004 = 3. EtherCAT command NOT sent (NOP requested)
	...
	0x4000 = 15. EtherCAT command NOT sent (NOP requested)
	0x8000 = complete frame NOT sent*)
	FR7WcState: UINT;
	(*
	0x0001 = wrong working counter of 1. EtherCAT command received
	0x0002 = wrong working counter of 2. EtherCAT command received
	0x0004 = wrong working counter of 3. EtherCAT command received
	...
	0x4000 = wrong working counter of 15. EtherCAT command received
	0x8000 = complete frame missing*)
	FR9State: UINT;
	(*
	0x0001 = 1. EtherCAT command NOT sent (NOP requested)
	0x0002 = 2. EtherCAT command NOT sent (NOP requested)
	0x0004 = 3. EtherCAT command NOT sent (NOP requested)
	...
	0x4000 = 15. EtherCAT command NOT sent (NOP requested)
	0x8000 = complete frame NOT sent*)
	FR9WcState: UINT;
	(*
	0x0001 = wrong working counter of 1. EtherCAT command received
	0x0002 = wrong working counter of 2. EtherCAT command received
	0x0004 = wrong working counter of 3. EtherCAT command received
	...
	0x4000 = wrong working counter of 15. EtherCAT command received
	0x8000 = complete frame missing*)

	SlaveCount: UINT;
	(*
	Actual count of EtherCAT slaves received*)

	DevState: UINT;
	(*
	0x0001 = Link error
	0x0002 = I/O locked after link error (I/O reset required)
	0x0004 = Link error (redundancy adapter)
	0x0008 = Missing one frame (redundancy mode)
	0x0010 = Out of send resources (I/O reset required)
	0x0020 = Watchdog triggered
	0x0040 = Ethernet driver (miniport) not found
	0x0080 = I/O reset active
	0x0100 = At least one device in 'INIT' state
	0x0200 = At least one device in 'PRE-OP' state
	0x0400 = At least one device in 'SAFE-OP' state
	0x0800 = At least one device indicates an error state
	0x1000 = DC not in sync*)

	CfgSlaveCount: UINT;
	(*
	Count of configured EtherCAT slaves
	*)
END_STRUCT
END_TYPE

// ---- Data types/Beckhoff IO udts/udt_ECATMaster_Status_20141211.TcDUT
(*udt (user defined type) of Beckhoff Type EtherCAT Master:
	auth. Brent Lekx-Toniolo of Toniolo Research & Development Inc.; 
	Version 1.0, July 2010
		- Initial Concept
	Version 20121206
		Changes from v1
			- Changed Interface to include Infodata udt Instance
			- Change to Naming Convention to include date as version
*)



TYPE udt_ECATMaster_Status_20141211 :
STRUCT
	Frm0State: UINT;
	(*
	0x0001 = 1. EtherCAT command NOT sent (NOP requested)
	0x0002 = 2. EtherCAT command NOT sent (NOP requested)
	0x0004 = 3. EtherCAT command NOT sent (NOP requested)
	...
	0x4000 = 15. EtherCAT command NOT sent (NOP requested)
	0x8000 = complete frame NOT sent*)
	Frm0WcState: UINT;
	(*
	0x0001 = wrong working counter of 1. EtherCAT command received
	0x0002 = wrong working counter of 2. EtherCAT command received
	0x0004 = wrong working counter of 3. EtherCAT command received
	...
	0x4000 = wrong working counter of 15. EtherCAT command received
	0x8000 = complete frame missing*)
	FR1State: UINT;
	(*
	0x0001 = 1. EtherCAT command NOT sent (NOP requested)
	0x0002 = 2. EtherCAT command NOT sent (NOP requested)
	0x0004 = 3. EtherCAT command NOT sent (NOP requested)
	...
	0x4000 = 15. EtherCAT command NOT sent (NOP requested)
	0x8000 = complete frame NOT sent*)
	FR1WcState: UINT;
	(*
	0x0001 = wrong working counter of 1. EtherCAT command received
	0x0002 = wrong working counter of 2. EtherCAT command received
	0x0004 = wrong working counter of 3. EtherCAT command received
	...
	0x4000 = wrong working counter of 15. EtherCAT command received
	0x8000 = complete frame missing*)
	FR2State: UINT;
	(*
	0x0001 = 1. EtherCAT command NOT sent (NOP requested)
	0x0002 = 2. EtherCAT command NOT sent (NOP requested)
	0x0004 = 3. EtherCAT command NOT sent (NOP requested)
	...
	0x4000 = 15. EtherCAT command NOT sent (NOP requested)
	0x8000 = complete frame NOT sent*)
	FR2WcState: UINT;
	(*
	0x0001 = wrong working counter of 1. EtherCAT command received
	0x0002 = wrong working counter of 2. EtherCAT command received
	0x0004 = wrong working counter of 3. EtherCAT command received
	...
	0x4000 = wrong working counter of 15. EtherCAT command received
	0x8000 = complete frame missing*)
	FR3State: UINT;
	(*
	0x0001 = 1. EtherCAT command NOT sent (NOP requested)
	0x0002 = 2. EtherCAT command NOT sent (NOP requested)
	0x0004 = 3. EtherCAT command NOT sent (NOP requested)
	...
	0x4000 = 15. EtherCAT command NOT sent (NOP requested)
	0x8000 = complete frame NOT sent*)
	FR3WcState: UINT;
	(*
	0x0001 = wrong working counter of 1. EtherCAT command received
	0x0002 = wrong working counter of 2. EtherCAT command received
	0x0004 = wrong working counter of 3. EtherCAT command received
	...
	0x4000 = wrong working counter of 15. EtherCAT command received
	0x8000 = complete frame missing*)
	FR4State: UINT;
	(*
	0x0001 = 1. EtherCAT command NOT sent (NOP requested)
	0x0002 = 2. EtherCAT command NOT sent (NOP requested)
	0x0004 = 3. EtherCAT command NOT sent (NOP requested)
	...
	0x4000 = 15. EtherCAT command NOT sent (NOP requested)
	0x8000 = complete frame NOT sent*)
	FR4WcState: UINT;
	(*
	0x0001 = wrong working counter of 1. EtherCAT command received
	0x0002 = wrong working counter of 2. EtherCAT command received
	0x0004 = wrong working counter of 3. EtherCAT command received
	...
	0x4000 = wrong working counter of 15. EtherCAT command received
	0x8000 = complete frame missing*)



	SlaveCount: UINT;
	(*
	Actual count of EtherCAT slaves received*)

	DevState: UINT;
	(*
	0x0001 = Link error
	0x0002 = I/O locked after link error (I/O reset required)
	0x0004 = Link error (redundancy adapter)
	0x0008 = Missing one frame (redundancy mode)
	0x0010 = Out of send resources (I/O reset required)
	0x0020 = Watchdog triggered
	0x0040 = Ethernet driver (miniport) not found
	0x0080 = I/O reset active
	0x0100 = At least one device in 'INIT' state
	0x0200 = At least one device in 'PRE-OP' state
	0x0400 = At least one device in 'SAFE-OP' state
	0x0800 = At least one device indicates an error state
	0x1000 = DC not in sync*)


	Infodata: udt_ECATMaster_InfoData_20121206;

END_STRUCT
END_TYPE

// ---- Data types/Beckhoff IO udts/udt_ECATSlave_Status.TcDUT
TYPE udt_ECATSlave_Status :
	STRUCT
		State: INT;
		(*
		0x___1 = Slave in 'INIT' state
		0x___2 = Slave in 'PREOP' state
		0x___3 = Slave in 'BOOT' state
		0x___4 = Slave in 'SAFEOP' state
		0x___8 = Slave in 'OP' state
		0x001_ = Slave signals error
		0x002_ = Invalid vendorId, productCode... read
		0x004_ = Initialization error occurred
		0x008_ = Slave disabled
		0x010_ = Slave NOT present
		0x020_ = Slave signals link error
		0x040_ = Slave signals missing link
		0x080_ = Slave signals unexpected link
		0x100_ = Communication port A
		0x200_ = Communication port B
		0x400_ = Communication port C
		0x800_ = Communication port D
		*)
	END_STRUCT
END_TYPE

// ---- Data types/Beckhoff IO udts/udt_ECATSlave_StatusADS.TcDUT
TYPE udt_ECATSlave_StatusADS :
	STRUCT
		State: INT;
		(*
		0x___1 = Slave in 'INIT' state
		0x___2 = Slave in 'PREOP' state
		0x___3 = Slave in 'BOOT' state
		0x___4 = Slave in 'SAFEOP' state
		0x___8 = Slave in 'OP' state
		0x001_ = Slave signals error
		0x002_ = Invalid vendorId, productCode... read
		0x004_ = Initialization error occurred
		0x008_ = Slave disabled
		0x010_ = Slave NOT present
		0x020_ = Slave signals link error
		0x040_ = Slave signals missing link
		0x080_ = Slave signals unexpected link
		0x100_ = Communication port A
		0x200_ = Communication port B
		0x400_ = Communication port C
		0x800_ = Communication port D
		*)

		AdsAddr_Port: UINT;

	END_STRUCT
END_TYPE

// ---- Data types/Beckhoff IO udts/udt_ECATSlave_StatusEXT.TcDUT
TYPE udt_ECATSlave_StatusEXT :
STRUCT
	State: UINT;
	(*
	0x___1 = Slave in 'INIT' state
	0x___2 = Slave in 'PREOP' state
	0x___3 = Slave in 'BOOT' state
	0x___4 = Slave in 'SAFEOP' state
	0x___8 = Slave in 'OP' state
	0x001_ = Slave signals error
	0x002_ = Invalid vendorId, productCode... read
	0x004_ = Initialization error occurred
	0x008_ = Slave disabled
	0x010_ = Slave NOT present
	0x020_ = Slave signals link error
	0x040_ = Slave signals missing link
	0x080_ = Slave signals unexpected link
	0x100_ = Communication port A
	0x200_ = Communication port B
	0x400_ = Communication port C
	0x800_ = Communication port D
	*)
	AdsAddr: udt_Generic_AdsAddr;
END_STRUCT
END_TYPE

// ---- Data types/Beckhoff IO udts/udt_ECATSlave_Status_CU1128.TcDUT
TYPE udt_ECATSlave_Status_CU1128 :
	STRUCT
		State: UINT;
		(*
		0x___1 = Slave in 'INIT' state
		0x___2 = Slave in 'PREOP' state
		0x___3 = Slave in 'BOOT' state
		0x___4 = Slave in 'SAFEOP' state
		0x___8 = Slave in 'OP' state
		0x001_ = Slave signals error
		0x002_ = Invalid vendorId, productCode... read
		0x004_ = Initialization error occurred
		0x008_ = Slave disabled
		0x010_ = Slave NOT present
		0x020_ = Slave signals link error
		0x040_ = Slave signals missing link
		0x080_ = Slave signals unexpected link
		0x100_ = Communication port A
		0x200_ = Communication port B
		0x400_ = Communication port C
		0x800_ = Communication port D
		*)
	END_STRUCT
END_TYPE

// ---- Data types/Beckhoff IO udts/udt_ECATSlave_Status_EP9128.TcDUT
TYPE udt_ECATSlave_Status_EP9128 :
	STRUCT
		State: UINT;
		(*
		0x___1 = Slave in 'INIT' state
		0x___2 = Slave in 'PREOP' state
		0x___3 = Slave in 'BOOT' state
		0x___4 = Slave in 'SAFEOP' state
		0x___8 = Slave in 'OP' state
		0x001_ = Slave signals error
		0x002_ = Invalid vendorId, productCode... read
		0x004_ = Initialization error occurred
		0x008_ = Slave disabled
		0x010_ = Slave NOT present
		0x020_ = Slave signals link error
		0x040_ = Slave signals missing link
		0x080_ = Slave signals unexpected link
		0x100_ = Communication port A
		0x200_ = Communication port B
		0x400_ = Communication port C
		0x800_ = Communication port D
		*)
	END_STRUCT
END_TYPE

// ---- Data types/Beckhoff IO udts/udt_EK1100.TcDUT
(*udt (user defined type) of Beckhoff EK1100 - EtherCAT Bus Coupler (Slave):
	auth. Brent Lekx-Toniolo of Toniolo Research & Development Inc.; 
	July 2010; version 1.0*)


TYPE udt_EK1100 :
STRUCT
 	InfoData: udt_ECATSlave_Status;
END_STRUCT
END_TYPE

// ---- Data types/Beckhoff IO udts/udt_EK1110_20150812.TcDUT
(*udt (user defined type) of Beckhoff EK1110 - EtherCAT ExtensionTerminal:
	
------------------------------------------------------------------------
REVISION NOTES:
	Original Author(s): b.lekx-toniolo
	Version 20150812
		- Initial Concept

------------------------------------------------------------------------
*)
TYPE udt_EK1110_20150812 :
STRUCT
	InfoData: udt_ECATSlave_Status;
END_STRUCT
END_TYPE

// ---- Data types/Beckhoff IO udts/udt_EK1122.TcDUT
(*udt (user defined type) of Beckhoff EK1122 - EtherCAT Junction Terminal:
	auth. Brent Lekx-Toniolo of Toniolo Research & Development Inc.; 
	July 2010; version 1.0*)

TYPE udt_EK1122 :
STRUCT
	InfoData: udt_ECATSlave_Status;
END_STRUCT
END_TYPE

// ---- Data types/Beckhoff IO udts/udt_EL1004.TcDUT
(*udt (user defined type) of Beckhoff EL1004 - 4 Point NPN/PNP Type Input Terminal:
	auth. Brent Lekx-Toniolo of Toniolo Research & Development Inc.; 
	July 2010; version 1.0*)


TYPE udt_EL1004 :
STRUCT
	I0: BOOL;				(*Input 0*)
	I1: BOOL;				(*Input 1*)
	I2: BOOL;				(*Input 2*)
	I3: BOOL;				(*Input 3*)
	InfoData: udt_ECATSlave_Status;
END_STRUCT
END_TYPE

// ---- Data types/Beckhoff IO udts/udt_EL1004_v2.TcDUT
(*udt (user defined type) of Beckhoff EL1004 - 4 Point NPN/PNP Type Input Terminal:
	auth. Brent Lekx-Toniolo of Toniolo Research & Development Inc.; 
	July 2010;
	Modified for tag reduction by R.Remillard
	November 2012; version 2.0*)


TYPE udt_EL1004_v2 :
STRUCT
	I: BYTE;				(*Input 0 - 3*)

	InfoData: udt_ECATSlave_Status;
END_STRUCT
END_TYPE

// ---- Data types/Beckhoff IO udts/udt_EL1008.TcDUT
(*udt (user defined type) of Beckhoff EL1008 Terminal, 8-channel digital input, 24 V DC, 3 ms
	auth. Brent Lekx-Toniolo of Toniolo Research & Development Inc.; 
	
------------------------------------------------------------------------
REVISION NOTES:
	Version 1.0: June 2023
		- Initial Concept, Copied From Original 6900 STAT, a. lopez

------------------------------------------------------------------------
*)


TYPE udt_EL1008 :
STRUCT
	I: BYTE;				(*Input 0 - 7*)

	InfoData: udt_ECATSlave_Status;
END_STRUCT
END_TYPE

// ---- Data types/Beckhoff IO udts/udt_EL1904.TcDUT
(*udt (user defined type) of Beckhoff EL1904 - 4 Point PNP Safety Type Input Terminal:
	auth. Brent Lekx-Toniolo of Toniolo Research & Development Inc.; 
	July 2010; version 1.0*)


TYPE udt_EL1904 :
STRUCT
	I0: BOOL;
	I1: BOOL;
	I2: BOOL;
	I3: BOOL;
	InfoData: udt_ECATSlave_Status;
END_STRUCT
END_TYPE

// ---- Data types/Beckhoff IO udts/udt_EL1904_v2.TcDUT
(*udt (user defined type) of Beckhoff EL1904 - 4 Point PNP Safety Type Input Terminal:
	auth. Brent Lekx-Toniolo of Toniolo Research & Development Inc.; 
	July 2010;
	Modified for tag reduction by R.Remillard
	November 2012; version 2.0*)


TYPE udt_EL1904_v2 :
STRUCT
	I: BYTE;

	InfoData: udt_ECATSlave_Status;
END_STRUCT
END_TYPE

// ---- Data types/Beckhoff IO udts/udt_EL2008.TcDUT
(*udt (user defined type) of Beckhoff EL2008 - 8 Point PNP Type Output Terminal:
	auth. Brent Lekx-Toniolo of Toniolo Research & Development Inc.; 
	July 2010;version 1.0*)


TYPE udt_EL2008 :
STRUCT
	Q0: BOOL;
	Q1: BOOL;
	Q2: BOOL;
	Q3: BOOL;
	Q4: BOOL;
	Q5: BOOL;
	Q6: BOOL;
	Q7: BOOL;
END_STRUCT
END_TYPE

// ---- Data types/Beckhoff IO udts/udt_EL2008_STAT.TcDUT
(*udt (user defined type) of Beckhoff EL2008 - 8 Point PNP Type Output Terminal:
	To work in conjunction of udt_EL2008
	auth. Brent Lekx-Toniolo of Toniolo Research & Development Inc.; 
	July 2010; version 1.0*)


TYPE udt_EL2008_STAT :
STRUCT
	InfoData: udt_ECATSlave_Status;
END_STRUCT
END_TYPE

// ---- Data types/Beckhoff IO udts/udt_EL2008_v2.TcDUT
(*udt (user defined type) of Beckhoff EL2008 - 8 Point PNP Type Output Terminal:
	auth. Brent Lekx-Toniolo of Toniolo Research & Development Inc.; 
	July 2010;
	Modified for tag reduction by R.Remillard
	November 2012; version 2.0*)


TYPE udt_EL2008_v2 :
STRUCT
	Q: BYTE;

END_STRUCT
END_TYPE

// ---- Data types/Beckhoff IO udts/udt_EL2622.TcDUT
(*udt (user defined type) of Beckhoff EL2622 - 2 Point Relay Type Output Terminal:
	auth. Brent Lekx-Toniolo of Toniolo Research & Development Inc.; 
	July 2010; version 1.0*)


TYPE udt_EL2622 :
STRUCT
	Q0: BOOL;
	Q1: BOOL;
END_STRUCT
END_TYPE

// ---- Data types/Beckhoff IO udts/udt_EL2622_STAT.TcDUT
(*udt (user defined type) of Beckhoff EL2622 - 2 Point Relay Type Output Terminal:
	To work in conjunction of udt_EL2008
	auth. Brent Lekx-Toniolo of Toniolo Research & Development Inc.; 
	July 2010; version 1.0*)


TYPE udt_EL2622_STAT :
STRUCT
	InfoData: udt_ECATSlave_Status;
END_STRUCT
END_TYPE

// ---- Data types/Beckhoff IO udts/udt_EL2904.TcDUT
(*udt (user defined type) of Beckhoff EL2904 - 4 Point PNP Safety Type Output Terminal:
	auth. Brent Lekx-Toniolo of Toniolo Research & Development Inc.; 
	July 2010; version 1.0*)


TYPE udt_EL2904 :
STRUCT
	Q0: BOOL;
	Q1: BOOL;
	Q2: BOOL;
	Q3: BOOL;
	InfoData: udt_ECATSlave_Status;
END_STRUCT
END_TYPE

// ---- Data types/Beckhoff IO udts/udt_EL2904RO.TcDUT
(*udt (user defined type) of Beckhoff EL2904 - 4 Point PNP Safety Type Output Terminal:
	auth. Brent Lekx-Toniolo of Toniolo Research & Development Inc.; 
	July 2010; version 1.0*)


TYPE udt_EL2904RO :
STRUCT
	Q0: BOOL;
	Q1: BOOL;
	Q2: BOOL;
	Q3: BOOL;
	InfoData: udt_ECATSlave_Status;
END_STRUCT
END_TYPE

// ---- Data types/Beckhoff IO udts/udt_EL2904RO_v2.TcDUT
(*udt (user defined type) of Beckhoff EL2904 - 4 Point PNP Safety Type Output Terminal:
	auth. Brent Lekx-Toniolo of Toniolo Research & Development Inc.; 
	July 2010;
	Modified for tag reduction by R.Remillard
	November 2012; version 2.0*)



TYPE udt_EL2904RO_v2 :
STRUCT
	Q: BYTE;

	InfoData: udt_ECATSlave_Status;
END_STRUCT
END_TYPE

// ---- Data types/Beckhoff IO udts/udt_EL3052.TcDUT
(*udt (user defined type) of Beckhoff EL3052 - 2 channel, 4 TO 20ma, Analog Input Terminal:
	auth. Brent Lekx-Toniolo of Toniolo Research & Development Inc.; 
	October July; version 1.0*)


TYPE udt_EL3052 :
STRUCT
	CH1: INT;
	CH2: INT;
	InfoData: udt_ECATSlave_Status;
END_STRUCT
END_TYPE

// ---- Data types/Beckhoff IO udts/udt_EL6692_20121204.TcDUT
(*udt (user defined type) of Beckhoff EL6692 - EtherCAT Bridge:
	auth. Brent Lekx-Toniolo of Sodecia GTAC.; 
	Version 1.0: November 2012
		- Initial Concept
	Version 20121204
		Changes from v1
			- Change to Naming Convention to include date as version

	Last Edit: December 4th, 2012, blt
*)

TYPE udt_EL6692_20121204 :
STRUCT
	SyncMode: UINT;
		(*	0: no Syncronisation
			1: Secondary side is Sync Master
			2: Primary side is Sync Master*)
	TxPDO_Toogle: BOOL;
		(*	Bit toggles when new data from other side received*)
	TxPDO_State: BOOL;
		(*	0: Other side is in OP state
			>0: Error*)
	Control_value_update_toggle: BOOL;
		(*	Bit toggles when new DC control data available*)
	Timestamp_update_toggle: BOOL;
		(*	 Bit toggles when new timestamp data available*)
	External_device_not_connected: BOOL;
		(*	0: External device connected
			1: External device not connected*)

	InfoData: udt_ECATSlave_Status;
END_STRUCT
END_TYPE

// ---- Data types/Beckhoff IO udts/udt_EL6695_20151028.TcDUT
(*udt (user defined type) of Beckhoff EL6695-1001 - EtherCAT Bridge (Specific to Kuka FSoE):
	auth. Brent Lekx-Toniolo of Sodecia GTAC.; 
	Version 20151028
		- initial concept, blt
*)

TYPE udt_EL6695_20151028 :
STRUCT

(*Data from Module 1, Sync Inputs*)
	TxPDO_Toogle: BOOL;
		(*	Bit toggles when new data from other side received*)
	TxPDO_State: BOOL;
		(*	0: Other side is in OP state
			>0: Error*)
	External_device_not_connected: BOOL;
		(*	0: External device connected
			1: External device not connected*)

(*Inputs and Outputs from Module 2, Safety Data*)
	FSOE_Inputs_Data_0: UINT;
	FSOE_Inputs_Data_1: UINT;
	FSOE_Inputs_Data_2: UINT;
	FSOE_Inputs_Data_3: UINT;
	FSOE_Inputs_ConnID: UINT;

	FSOE_Outputs_Data_0: UINT;
	FSOE_Outputs_Data_1: UINT;
	FSOE_Outputs_Data_2: UINT;
	FSOE_Outputs_Data_3: UINT;


	InfoData: udt_ECATSlave_StatusEXT;
END_STRUCT
END_TYPE

// ---- Data types/Beckhoff IO udts/udt_EL6731.TcDUT
(*udt (user defined type) of Beckhoff EL6731 - Profibus Mater, ECAT Terminal:
	auth. Brent Lekx-Toniolo of Toniolo Research & Development Inc.; 
	July 2010; version 1.0*)


TYPE udt_EL6731 :
STRUCT
	Error: USINT;
	(*Error:
	 indicates the number of boxes with a BoxState unequal zero*)
	Wc_State: BOOL;
	(*0 = Data valid
	1 = Data invalid*)
	InfoData: udt_ECATSlave_Status;
END_STRUCT
END_TYPE

// ---- Data types/Beckhoff IO udts/udt_EL6900_CMD.TcDUT
(*udt (user defined type) of Beckhoff EL6900 - TwinSAFE Controller:
	auth. Brent Lekx-Toniolo of Toniolo Research & Development Inc.; 
	July 2010; version 1.0*)

TYPE udt_EL6900_CMD :
	STRUCT
	SG: ARRAY[0..7] OF udt_EL6900_SafetyGroup_CMD;
	END_STRUCT
END_TYPE

// ---- Data types/Beckhoff IO udts/udt_EL6900_CMD_20121204.TcDUT
(*udt (user defined type) of Beckhoff EL6900 - TwinSAFE Controller Command Interface:
	auth: Brent Lekx-Toniolo/Rob Remillard of Sodecia GTAC
	Version 1.0: November 2012
		- Initial Concept
	Version 20121204
		Changes from v1
			- Change to Naming Convention to include date as version

	Last Edit: December 4th, 2012, blt
*)


TYPE udt_EL6900_CMD_20121204 :
	STRUCT
	SGs_RUNSTOP: BOOL;
	(*
	RUN/STOP for all Safety Groups in Terminal*)

	SGs_ERRAck: BOOL;
	(*
	ERR Ack for all Safety Groups in Terminal*)

	FBs_ControlPowerPB: BOOL;
	(*
	Reset from Control Power  for all FBs in Terminal*)

	FBs_Restart_Spare: BOOL;
	(*
	Spare Reset for future use by FBs in Terminal*)


	END_STRUCT
END_TYPE

// ---- Data types/Beckhoff IO udts/udt_EL6900_DeviceInfoData_20160426.TcDUT
(*udt (user defined type) Device Info Data Section (configurable) of Beckhoff EL6900 - TwinSAFE Controller
	auth. Brent Lekx-Toniolo of Sodecia GTAC.; 
------------------------------------------------------------------------
REVISION NOTES:
	Version 20160426
			- Original Concept, b.lekx-toniolo

------------------------------------------------------------------------

*)



TYPE udt_EL6900_DeviceInfoData_20160426 :
	STRUCT
		(*Project CRC*)
		Project_CRC: UINT;

	END_STRUCT
END_TYPE

// ---- Data types/Beckhoff IO udts/udt_EL6900_SafetyGroup_CMD.TcDUT
TYPE udt_EL6900_SafetyGroup_CMD :
	STRUCT
	Run_Stop: BOOL;
	Error_Ack: BOOL;
	FB_Restart: ARRAY[0..31] OF BOOL;
	END_STRUCT
END_TYPE

// ---- Data types/Beckhoff IO udts/udt_EL6900_SafetyGroup_STAT.TcDUT
(*udt (user defined type) of Beckhoff EL6900 - TwinSAFE Controller:
	auth. Brent Lekx-Toniolo of Toniolo Research & Development Inc.; 
	July 2010; version 1.0*)

TYPE udt_EL6900_SafetyGroup_STAT :
	STRUCT
	FB_In_Error: BOOL;
	Com_Error: BOOL;
	Out_Error: BOOL;
	FB_Error: ARRAY[0..31] OF BOOL;

	END_STRUCT
END_TYPE

// ---- Data types/Beckhoff IO udts/udt_EL6900_STAT.TcDUT
(*udt (user defined type) of Beckhoff EL6900 - TwinSAFE Controller:
	auth. Brent Lekx-Toniolo of Toniolo Research & Development Inc.; 
	July 2010; version 1.0*)

TYPE udt_EL6900_STAT :
	STRUCT
	SG: ARRAY[0..7] OF udt_EL6900_SafetyGroup_STAT;
	InfoData: udt_ECATSlave_Status;

	END_STRUCT
END_TYPE

// ---- Data types/Beckhoff IO udts/udt_EL6900_STAT_20160426.TcDUT
(*udt (user defined type) of Beckhoff EL6900 - TwinSAFE Controller Status Interface:
	auth. Brent Lekx-Toniolo/Rob Remillard of Sodecia GTAC.; 
------------------------------------------------------------------------
REVISION NOTES:
	Version 1.0: November 2012
		- Initial Concept
	Version 20121204
		Changes from v1
			- Change to Naming Convention to include date as version
	Version 20150925
			- Added variable for area to store terminal temperature data, b.lekx-toniolo
			- Changed InfoData to EX type to allow linking area for AMS and Port, b.lekx-toniolo
	Version 20160426
			- Added Instance of udt_EL6900_DeviceInfoData_yyyymmdd, b.lekx-toniolo

------------------------------------------------------------------------

*)

TYPE udt_EL6900_STAT_20160426 :
	STRUCT
	SGs_FB_ERR: BYTE;
	(*
	FB ERROR Status Summary of ALL FBs in Terminal, 1 bit per SG*)

	SGs_COM_ERR: BYTE;
	(*
	COM Status of all Coms Linked to Terminal, 1 bit per SG*)

	SGs_OUT_ERR: BYTE;
	(*
	OUTPUT ERROR Status of all Outputs Linked to Terminal, 1 bit per SG*)

	FBs_FB_ERR: DINT;
	(*
	FB ERROR Status fof EACH FB within Terminal, 1 bit per FB*)

	Device_Info_Data: udt_EL6900_DeviceInfoData_20160426;
	InfoData: udt_ECATSlave_StatusEXT;

	(*CoE Data Section*)
	CoE_Project_State:	UDINT;	(*Retreived via CoE - For Storage of Safety Project State*)
	CoE_Temperature_1: 	UINT; 	(*Retreived via CoE - For Storage of Primary Temperature MC1 Data*)
	CoE_Temperature_2: 	UINT;  	(*Retreived via CoE - For Storage of Secondary Temperature MC1 Data*)


	END_STRUCT
END_TYPE

// ---- Data types/Beckhoff IO udts/udt_EL94xx.TcDUT
(*udt (user defined type) of Beckhoff EL94xx - Ebus Power Terminal:
	auth. Brent Lekx-Toniolo of Toniolo Research & Development Inc.; 
	July 2010; version 1.0*)


TYPE udt_EL94xx :
STRUCT
	Us_Undervoltage: BOOL;
	Up_UnderVoltage: BOOL;
	WcState: BOOL;
	(*0 = Data valid
	1 = Data invalid*)
	InfoData: udt_ECATSlave_Status;
END_STRUCT
END_TYPE

// ---- Data types/Beckhoff IO udts/udt_EP1008_002.TcDUT
(*udt (user defined type) of Beckhoff EP1008-0002 - 8 Point IP67 Rated Digital Input Box:
	auth. Brent Lekx-Toniolo of Toniolo Research & Development Inc.; 
	July 2010; version 1.0*)


TYPE udt_EP1008_002 :
STRUCT
	I0: BOOL;
	I1: BOOL;
	I2: BOOL;
	I3: BOOL;
	I4: BOOL;
	I5: BOOL;
	I6: BOOL;
	I7: BOOL;
	Wc_State: BOOL;
	(*0 = Data valid
	1 = Data invalid*)
	InfoData: udt_ECATSlave_Status;
END_STRUCT
END_TYPE

// ---- Data types/Beckhoff IO udts/udt_EP1008_002_v2.TcDUT
(*udt (user defined type) of Beckhoff EP1008-0002 - 8 Point IP67 Rated Digital Input Box:
	auth. Brent Lekx-Toniolo of Toniolo Research & Development Inc.; 
	July 2010;
	Modified for tag reduction by R.Remillard
	November 2012; version 2.0*)


TYPE udt_EP1008_002_v2 :
STRUCT
	I: BYTE;						(*Use a single BYTE to replace the 8 BOOLs to reduce the # of tags*)

	Wc_State: BOOL;
	(*0 = Data valid
	1 = Data invalid*)
	InfoData: udt_ECATSlave_Status;
END_STRUCT
END_TYPE

// ---- Data types/Beckhoff IO udts/udt_EP1111.TcDUT
(*udt (user defined type) of Beckhoff EP1111 -  IP67 Rated ID Box:
	auth. Rob Remillard; 
	March 2014;*)


TYPE udt_EP1111 :
STRUCT
	ID: UINT;

	Wc_State: BOOL;
	(*0 = Data valid
	1 = Data invalid*)
	InfoData: udt_ECATSlave_Status;
END_STRUCT
END_TYPE

// ---- Data types/Beckhoff IO udts/udt_EP1908_002.TcDUT
(*udt (user defined type) of Beckhoff EL1908 - 8 Point PNP Safety Type Input Terminal:
	June 2014;*)


TYPE udt_EP1908_002 :
STRUCT
	I: BYTE;

	InfoData: udt_ECATSlave_Status;
END_STRUCT
END_TYPE

// ---- Data types/Beckhoff IO udts/udt_EP1918.TcDUT
(*udt (user defined type) of Beckhoff Ep1918 - EtherCAT Bus Coupler (Slave):
	auth. Brent Lekx-Toniolo of Toniolo Research & Development Inc.; 
	April 2025; version 1.0 - created, r.jones*)


TYPE udt_EP1918 :
STRUCT
	I AT %I*: BYTE;
	STAT AT %I*: udt_EP1918_STAT_20250213;
	CMD AT %Q*: udt_EP1918_CMD_20250213;
	InfoData: udt_ECATSlave_Status;
	NotPresent: BOOL;
	PortB_MissingLink: BOOL;
	
END_STRUCT
END_TYPE

// ---- Data types/Beckhoff IO udts/udt_EP1918_CMD_20250213.TcDUT
(*udt (user defined type) of Beckhoff EL6900 - TwinSAFE Controller Command Interface:
	auth: Brent Lekx-Toniolo/Rob Remillard of Sodecia GTAC
	Version 1.0: November 2012
		- Initial Concept
	Version 20121204
		Changes from v1
			- Change to Naming Convention to include date as version

	Last Edit: December 4th, 2012, blt
*)


TYPE udt_EP1918_CMD_20250213 :
	STRUCT
	SGs_RUNSTOP: BOOL;
	(*
	RUN/STOP for all Safety Groups in Terminal*)

	SGs_ERRAck: BOOL;
	(*
	ERR Ack for all Safety Groups in Terminal*)

	FBs_ControlPowerPB: BOOL;
	(*
	Reset from Control Power  for all FBs in Terminal*)

	FBs_Restart_Spare: BOOL;
	(*
	Spare Reset for future use by FBs in Terminal*)


	END_STRUCT
END_TYPE

// ---- Data types/Beckhoff IO udts/udt_EP1918_STAT_20250213.TcDUT
(*udt (user defined type) of Beckhoff EL6900 - TwinSAFE Controller Status Interface:
	auth. Brent Lekx-Toniolo/Rob Remillard of Sodecia GTAC.; 
------------------------------------------------------------------------
REVISION NOTES:
	Version 1.0: November 2012
		- Initial Concept
	Version 20121204
		Changes from v1
			- Change to Naming Convention to include date as version
	Version 20150925
			- Added variable for area to store terminal temperature data, b.lekx-toniolo
			- Changed InfoData to EX type to allow linking area for AMS and Port, b.lekx-toniolo
	Version 20160426
			- Added Instance of udt_EL6900_DeviceInfoData_yyyymmdd, b.lekx-toniolo

------------------------------------------------------------------------

*)

TYPE udt_EP1918_STAT_20250213 :
	STRUCT
	SGs_FB_ERR: BYTE;
	(*
	FB ERROR Status Summary of ALL FBs in Terminal, 1 bit per SG*)

	SGs_COM_ERR: BYTE;
	(*
	COM Status of all Coms Linked to Terminal, 1 bit per SG*)

	SGs_OUT_ERR: BYTE;
	(*
	OUTPUT ERROR Status of all Outputs Linked to Terminal, 1 bit per SG*)

	FBs_FB_ERR: DINT;
	(*
	FB ERROR Status fof EACH FB within Terminal, 1 bit per FB*)

	I: BYTE;

	Device_Info_Data: udt_EL6900_DeviceInfoData_20160426;
	InfoData: udt_ECATSlave_StatusEXT;

	(*CoE Data Section*)
	CoE_Project_State:	UDINT;	(*Retreived via CoE - For Storage of Safety Project State*)
	CoE_Temperature_1: 	UINT; 	(*Retreived via CoE - For Storage of Primary Temperature MC1 Data*)
	CoE_Temperature_2: 	UINT;  	(*Retreived via CoE - For Storage of Secondary Temperature MC1 Data*)


	END_STRUCT
END_TYPE

// ---- Data types/Beckhoff IO udts/udt_EP2028_002.TcDUT
(*udt (user defined type) of Beckhoff EP2028-0002 - 8 Point IP67 Rated Digital Output Box:
	auth. Brent Lekx-Toniolo of Toniolo Research & Development Inc.; 
	July 2010; version 1.0*)


TYPE udt_EP2028_002 :
STRUCT
	Q0: BOOL;
	Q1: BOOL;
	Q2: BOOL;
	Q3: BOOL;
	Q4: BOOL;
	Q5: BOOL;
	Q6: BOOL;
	Q7: BOOL;
END_STRUCT
END_TYPE

// ---- Data types/Beckhoff IO udts/udt_EP2028_002_STAT.TcDUT
(*udt (user defined type) of Beckhoff EP2028-002 IP67 Block - 8 Point Output Block:
	To work in conjunction of udt_EL2028_002
	auth. Brent Lekx-Toniolo of Toniolo Research & Development Inc.; 
	August 2010; version 1.0*)


TYPE udt_EP2028_002_STAT :
STRUCT
	InfoData: udt_ECATSlave_Status;
END_STRUCT
END_TYPE

// ---- Data types/Beckhoff IO udts/udt_EP2028_002_v2.TcDUT
(*udt (user defined type) of Beckhoff EP2028-0002 - 8 Point IP67 Rated Digital Output Box:
	auth. Brent Lekx-Toniolo of Toniolo Research & Development Inc.; 
	July 2010;
	Modified for tag reduction by R.Remillard
	November 2012; version 2.0*)


TYPE udt_EP2028_002_v2 :
STRUCT
	Q: BYTE;

END_STRUCT
END_TYPE

